Universal Robots URScript: 2024golden.script

def unnamed():
  set_tcp(p[0.0,0.0,0.0,0.0,0.0,0.0])
  set_standard_analog_input_domain(0, 1)
  set_standard_analog_input_domain(1, 1)
  set_tool_analog_input_domain(0, 1)
  set_tool_analog_input_domain(1, 1)
  set_analog_outputdomain(0, 0)
  set_analog_outputdomain(1, 0)
  set_input_actions_to_default()
  set_target_payload(1.070000, [0.002000, 0.003000, 0.057000], [0.001723, 0.001723, 0.001723, 0.000000, 0.000000, 0.000000])
  set_tool_communication(True, 1000000, 2, 1, 1.5, 3.5)
  set_tool_output_mode(0)
  set_tool_digital_output_mode(0, 1)
  set_tool_digital_output_mode(1, 1)
  set_tool_voltage(0)
  set_gravity([0.0, 0.0, 9.82])
  step_count_2c8ba0bd_3175_4124_8579_105621cd2361 = 0.0
  thread Step_Counter_Thread_abff76f1_d808_4649_b515_a114c75a653f():
    while (True):
      step_count_2c8ba0bd_3175_4124_8579_105621cd2361 = step_count_2c8ba0bd_3175_4124_8579_105621cd2361 + 1.0
      sync()
    end
  end
  run Step_Counter_Thread_abff76f1_d808_4649_b515_a114c75a653f()
  set_safety_mode_transition_hardness(1)
  global Plane_1=p[-0.700006141123905,1.3454883874109249E-6,0.3910559577028425,-1.2089868272251132,-1.2089999932245832,1.20858562628424]
  global Plane_2=p[0.0,0.0,0.0,0.0,0.0,0.0]
  global Point_1=p[0.6913645118948067,-0.12399382748223003,0.49223711947071,-1.2983729986843258,1.1259514972191385,-1.2203503861141718]
  $ 1 "Robot Program"
  $ 2 "Script: 2024Dragon_V2_golden_pen.script"
  def Machining1():
    # Default parameters:
    global speed_ms = 0.3
    global speed_rads = 0.75
    global accel_mss = 3
    global accel_radss = 1.2
    global blend_radius_m = 0.001

    # Add subprograms here
    # Start of main program
    # Program generated by RoboDK v5.6.5 for UR10e on 10/01/2024 17:37:16
    # Using nominal kinematics.
    blend_radius_m = 0.001
    speed_ms = 1.000
    # set_reference(p[0.320000, -0.152000, -0.013500, 0.000000, 0.000000, 0.000000])
    set_tcp(p[0.000000, 0.000000, 0.252000, 0.000000, 0.000000, 0.000000])
    # Show Tool
    movej([0.070455, -1.056852, -2.625487, -1.030050, 1.570796, 1.641252],accel_radss,speed_rads,0,blend_radius_m)
    movel([0.070455, -1.056852, -2.625487, -1.030050, 1.570796, 1.641252],accel_mss,speed_ms,0,blend_radius_m)
    # Splitting Linear movement in 32 (instruction 7: MoveL 3)
    movel([0.070455, -1.058454, -2.626785, -1.027150, 1.570796, 1.641252],accel_mss,speed_ms,0,blend_radius_m)
    movel([0.070455, -1.060067, -2.628081, -1.024241, 1.570796, 1.641252],accel_mss,speed_ms,0,blend_radius_m)
    movel([0.070455, -1.061692, -2.629375, -1.021322, 1.570796, 1.641252],accel_mss,speed_ms,0,blend_radius_m)
    movel([0.070455, -1.063329, -2.630667, -1.018394, 1.570796, 1.641252],accel_mss,speed_ms,0,blend_radius_m)
    movel([0.070455, -1.064977, -2.631956, -1.015456, 1.570796, 1.641252],accel_mss,speed_ms,0,blend_radius_m)
    movel([0.070455, -1.066637, -2.633243, -1.012509, 1.570796, 1.641252],accel_mss,speed_ms,0,blend_radius_m)
    movel([0.070455, -1.068308, -2.634528, -1.009553, 1.570796, 1.641252],accel_mss,speed_ms,0,blend_radius_m)
    movel([0.070455, -1.069991, -2.635811, -1.006586, 1.570796, 1.641252],accel_mss,speed_ms,0,blend_radius_m)
    movel([0.070455, -1.071686, -2.637092, -1.003611, 1.570796, 1.641252],accel_mss,speed_ms,0,blend_radius_m)
    movel([0.070455, -1.073393, -2.638371, -1.000625, 1.570796, 1.641252],accel_mss,speed_ms,0,blend_radius_m)
    movel([0.070455, -1.075112, -2.639647, -0.997630, 1.570796, 1.641252],accel_mss,speed_ms,0,blend_radius_m)
    movel([0.070455, -1.076843, -2.640921, -0.994625, 1.570796, 1.641252],accel_mss,speed_ms,0,blend_radius_m)
    movel([0.070455, -1.078586, -2.642192, -0.991611, 1.570796, 1.641252],accel_mss,speed_ms,0,blend_radius_m)
    movel([0.070455, -1.080341, -2.643462, -0.988586, 1.570796, 1.641252],accel_mss,speed_ms,0,blend_radius_m)
    movel([0.070455, -1.082109, -2.644729, -0.985551, 1.570796, 1.641252],accel_mss,speed_ms,0,blend_radius_m)
    movel([0.070455, -1.083888, -2.645994, -0.982507, 1.570796, 1.641252],accel_mss,speed_ms,0,blend_radius_m)
    movel([0.070455, -1.085680, -2.647256, -0.979453, 1.570796, 1.641252],accel_mss,speed_ms,0,blend_radius_m)
    movel([0.070455, -1.087485, -2.648516, -0.976388, 1.570796, 1.641252],accel_mss,speed_ms,0,blend_radius_m)
    movel([0.070455, -1.089301, -2.649774, -0.973313, 1.570796, 1.641252],accel_mss,speed_ms,0,blend_radius_m)
    movel([0.070455, -1.091131, -2.651030, -0.970229, 1.570796, 1.641252],accel_mss,speed_ms,0,blend_radius_m)
    movel([0.070455, -1.092973, -2.652283, -0.967134, 1.570796, 1.641252],accel_mss,speed_ms,0,blend_radius_m)
    movel([0.070455, -1.094827, -2.653533, -0.964028, 1.570796, 1.641252],accel_mss,speed_ms,0,blend_radius_m)
    movel([0.070455, -1.096695, -2.654781, -0.960913, 1.570796, 1.641252],accel_mss,speed_ms,0,blend_radius_m)
    movel([0.070455, -1.098575, -2.656027, -0.957787, 1.570796, 1.641252],accel_mss,speed_ms,0,blend_radius_m)
    movel([0.070455, -1.100468, -2.657271, -0.954651, 1.570796, 1.641252],accel_mss,speed_ms,0,blend_radius_m)
    movel([0.070455, -1.102374, -2.658511, -0.951504, 1.570796, 1.641252],accel_mss,speed_ms,0,blend_radius_m)
    movel([0.070455, -1.104293, -2.659750, -0.948346, 1.570796, 1.641252],accel_mss,speed_ms,0,blend_radius_m)
    movel([0.070455, -1.106224, -2.660986, -0.945179, 1.570796, 1.641252],accel_mss,speed_ms,0,blend_radius_m)
    movel([0.070455, -1.108170, -2.662219, -0.942000, 1.570796, 1.641252],accel_mss,speed_ms,0,blend_radius_m)
    movel([0.070455, -1.110128, -2.663450, -0.938811, 1.570796, 1.641252],accel_mss,speed_ms,0,blend_radius_m)
    movel([0.070455, -1.112099, -2.664678, -0.935611, 1.570796, 1.641252],accel_mss,speed_ms,0,blend_radius_m)
    movel([0.070455, -1.114084, -2.665904, -0.932401, 1.570796, 1.641252],accel_mss,speed_ms,0,blend_radius_m)
    movel([0.070455, -1.114084, -2.665904, -0.932401, 1.570796, 1.641252],accel_mss,speed_ms,0,blend_radius_m)
    speed_ms = 1.000
    movel([0.070455, -1.114084, -2.665904, -0.932401, 1.570796, 1.641252],accel_mss,speed_ms,0,blend_radius_m)
    movel([0.070455, -1.114084, -2.665904, -0.932401, 1.570796, 1.641252],accel_mss,speed_ms,0,blend_radius_m)
    movel([0.070455, -1.114084, -2.665904, -0.932401, 1.570796, 1.641252],accel_mss,speed_ms,0,blend_radius_m)
    speed_ms = 0.005
    # Splitting Linear movement in 22 (instruction 14: MoveL 8)
    movel([0.070455, -1.112159, -2.664716, -0.935514, 1.570796, 1.641252],accel_mss,speed_ms,0,blend_radius_m)
    movel([0.070455, -1.110247, -2.663525, -0.938618, 1.570796, 1.641252],accel_mss,speed_ms,0,blend_radius_m)
    movel([0.070455, -1.108347, -2.662331, -0.941711, 1.570796, 1.641252],accel_mss,speed_ms,0,blend_radius_m)
    movel([0.070455, -1.106460, -2.661135, -0.944794, 1.570796, 1.641252],accel_mss,speed_ms,0,blend_radius_m)
    movel([0.070455, -1.104584, -2.659937, -0.947867, 1.570796, 1.641252],accel_mss,speed_ms,0,blend_radius_m)
    movel([0.070455, -1.102722, -2.658737, -0.950930, 1.570796, 1.641252],accel_mss,speed_ms,0,blend_radius_m)
    movel([0.070455, -1.100871, -2.657534, -0.953984, 1.570796, 1.641252],accel_mss,speed_ms,0,blend_radius_m)
    movel([0.070455, -1.099033, -2.656329, -0.957027, 1.570796, 1.641252],accel_mss,speed_ms,0,blend_radius_m)
    movel([0.070455, -1.097206, -2.655121, -0.960061, 1.570796, 1.641252],accel_mss,speed_ms,0,blend_radius_m)
    movel([0.070455, -1.095392, -2.653912, -0.963085, 1.570796, 1.641252],accel_mss,speed_ms,0,blend_radius_m)
    movel([0.070455, -1.093590, -2.652700, -0.966100, 1.570796, 1.641252],accel_mss,speed_ms,0,blend_radius_m)
    movel([0.070455, -1.091799, -2.651486, -0.969104, 1.570796, 1.641252],accel_mss,speed_ms,0,blend_radius_m)
    movel([0.070455, -1.090021, -2.650269, -0.972099, 1.570796, 1.641252],accel_mss,speed_ms,0,blend_radius_m)
    movel([0.070455, -1.088254, -2.649050, -0.975085, 1.570796, 1.641252],accel_mss,speed_ms,0,blend_radius_m)
    movel([0.070455, -1.086499, -2.647829, -0.978061, 1.570796, 1.641252],accel_mss,speed_ms,0,blend_radius_m)
    movel([0.070455, -1.084755, -2.646606, -0.981027, 1.570796, 1.641252],accel_mss,speed_ms,0,blend_radius_m)
    movel([0.070455, -1.083024, -2.645381, -0.983984, 1.570796, 1.641252],accel_mss,speed_ms,0,blend_radius_m)
    movel([0.070455, -1.081304, -2.644153, -0.986932, 1.570796, 1.641252],accel_mss,speed_ms,0,blend_radius_m)
    movel([0.070455, -1.079595, -2.642924, -0.989870, 1.570796, 1.641252],accel_mss,speed_ms,0,blend_radius_m)
    movel([0.070455, -1.077898, -2.641692, -0.992799, 1.570796, 1.641252],accel_mss,speed_ms,0,blend_radius_m)
    movel([0.070455, -1.076212, -2.640458, -0.995719, 1.570796, 1.641252],accel_mss,speed_ms,0,blend_radius_m)
    movel([0.070455, -1.074538, -2.639222, -0.998630, 1.570796, 1.641252],accel_mss,speed_ms,0,blend_radius_m)
    speed_ms = 1.000
    # Splitting Linear movement in 22 (instruction 16: MoveL 9)
    movel([0.070455, -1.076212, -2.640458, -0.995719, 1.570796, 1.641252],accel_mss,speed_ms,0,blend_radius_m)
    movel([0.070455, -1.077898, -2.641692, -0.992799, 1.570796, 1.641252],accel_mss,speed_ms,0,blend_radius_m)
    movel([0.070455, -1.079595, -2.642924, -0.989870, 1.570796, 1.641252],accel_mss,speed_ms,0,blend_radius_m)
    movel([0.070455, -1.081304, -2.644153, -0.986932, 1.570796, 1.641252],accel_mss,speed_ms,0,blend_radius_m)
    movel([0.070455, -1.083024, -2.645381, -0.983984, 1.570796, 1.641252],accel_mss,speed_ms,0,blend_radius_m)
    movel([0.070455, -1.084755, -2.646606, -0.981027, 1.570796, 1.641252],accel_mss,speed_ms,0,blend_radius_m)
    movel([0.070455, -1.086499, -2.647829, -0.978061, 1.570796, 1.641252],accel_mss,speed_ms,0,blend_radius_m)
    movel([0.070455, -1.088254, -2.649050, -0.975085, 1.570796, 1.641252],accel_mss,speed_ms,0,blend_radius_m)
    movel([0.070455, -1.090021, -2.650269, -0.972099, 1.570796, 1.641252],accel_mss,speed_ms,0,blend_radius_m)
    movel([0.070455, -1.091799, -2.651486, -0.969104, 1.570796, 1.641252],accel_mss,speed_ms,0,blend_radius_m)
    movel([0.070455, -1.093590, -2.652700, -0.966100, 1.570796, 1.641252],accel_mss,speed_ms,0,blend_radius_m)
    movel([0.070455, -1.095392, -2.653912, -0.963085, 1.570796, 1.641252],accel_mss,speed_ms,0,blend_radius_m)
    movel([0.070455, -1.097206, -2.655121, -0.960061, 1.570796, 1.641252],accel_mss,speed_ms,0,blend_radius_m)
    movel([0.070455, -1.099033, -2.656329, -0.957027, 1.570796, 1.641252],accel_mss,speed_ms,0,blend_radius_m)
    movel([0.070455, -1.100871, -2.657534, -0.953984, 1.570796, 1.641252],accel_mss,speed_ms,0,blend_radius_m)
    movel([0.070455, -1.102722, -2.658737, -0.950930, 1.570796, 1.641252],accel_mss,speed_ms,0,blend_radius_m)
    movel([0.070455, -1.104584, -2.659937, -0.947867, 1.570796, 1.641252],accel_mss,speed_ms,0,blend_radius_m)
    movel([0.070455, -1.106460, -2.661135, -0.944794, 1.570796, 1.641252],accel_mss,speed_ms,0,blend_radius_m)
    movel([0.070455, -1.108347, -2.662331, -0.941711, 1.570796, 1.641252],accel_mss,speed_ms,0,blend_radius_m)
    movel([0.070455, -1.110247, -2.663525, -0.938618, 1.570796, 1.641252],accel_mss,speed_ms,0,blend_radius_m)
    movel([0.070455, -1.112159, -2.664716, -0.935514, 1.570796, 1.641252],accel_mss,speed_ms,0,blend_radius_m)
    movel([0.070455, -1.114084, -2.665904, -0.932401, 1.570796, 1.641252],accel_mss,speed_ms,0,blend_radius_m)
    speed_ms = 0.040
    movel([0.070455, -1.114084, -2.665904, -0.932401, 1.570796, 1.641252],accel_mss,speed_ms,0,blend_radius_m)
    speed_ms = 1.000
    movel([0.070455, -1.114084, -2.665904, -0.932401, 1.570796, 1.641252],accel_mss,speed_ms,0,blend_radius_m)
    # Splitting Linear movement in 152 (instruction 21: MoveL 12)
    movel([0.070832, -1.116719, -2.664817, -0.930853, 1.570796, 1.641628],accel_mss,speed_ms,0,blend_radius_m)
    movel([0.071206, -1.119347, -2.663727, -0.929315, 1.570796, 1.642002],accel_mss,speed_ms,0,blend_radius_m)
    movel([0.071578, -1.121968, -2.662633, -0.927788, 1.570796, 1.642374],accel_mss,speed_ms,0,blend_radius_m)
    movel([0.071947, -1.124581, -2.661536, -0.926272, 1.570796, 1.642743],accel_mss,speed_ms,0,blend_radius_m)
    movel([0.072314, -1.127187, -2.660435, -0.924767, 1.570796, 1.643111],accel_mss,speed_ms,0,blend_radius_m)
    movel([0.072679, -1.129786, -2.659331, -0.923272, 1.570796, 1.643476],accel_mss,speed_ms,0,blend_radius_m)
    movel([0.073042, -1.132378, -2.658223, -0.921788, 1.570796, 1.643839],accel_mss,speed_ms,0,blend_radius_m)
    movel([0.073403, -1.134962, -2.657112, -0.920315, 1.570796, 1.644199],accel_mss,speed_ms,0,blend_radius_m)
    movel([0.073761, -1.137540, -2.655997, -0.918852, 1.570796, 1.644558],accel_mss,speed_ms,0,blend_radius_m)
    movel([0.074117, -1.140110, -2.654879, -0.917400, 1.570796, 1.644914],accel_mss,speed_ms,0,blend_radius_m)
    movel([0.074472, -1.142673, -2.653758, -0.915958, 1.570796, 1.645268],accel_mss,speed_ms,0,blend_radius_m)
    movel([0.074824, -1.145229, -2.652633, -0.914527, 1.570796, 1.645620],accel_mss,speed_ms,0,blend_radius_m)
    movel([0.075173, -1.147778, -2.651505, -0.913106, 1.570796, 1.645970],accel_mss,speed_ms,0,blend_radius_m)
    movel([0.075521, -1.150320, -2.650374, -0.911695, 1.570796, 1.646318],accel_mss,speed_ms,0,blend_radius_m)
    movel([0.075867, -1.152855, -2.649239, -0.910295, 1.570796, 1.646663],accel_mss,speed_ms,0,blend_radius_m)
    movel([0.076211, -1.155382, -2.648101, -0.908905, 1.570796, 1.647007],accel_mss,speed_ms,0,blend_radius_m)
    movel([0.076552, -1.157903, -2.646960, -0.907526, 1.570796, 1.647349],accel_mss,speed_ms,0,blend_radius_m)
    movel([0.076892, -1.160417, -2.645816, -0.906157, 1.570796, 1.647688],accel_mss,speed_ms,0,blend_radius_m)
    movel([0.077230, -1.162924, -2.644668, -0.904797, 1.570796, 1.648026],accel_mss,speed_ms,0,blend_radius_m)
    movel([0.077565, -1.165423, -2.643517, -0.903448, 1.570796, 1.648362],accel_mss,speed_ms,0,blend_radius_m)
    movel([0.077899, -1.167916, -2.642363, -0.902110, 1.570796, 1.648695],accel_mss,speed_ms,0,blend_radius_m)
    movel([0.078231, -1.170402, -2.641206, -0.900781, 1.570796, 1.649027],accel_mss,speed_ms,0,blend_radius_m)
    movel([0.078561, -1.172882, -2.640045, -0.899462, 1.570796, 1.649357],accel_mss,speed_ms,0,blend_radius_m)
    movel([0.078888, -1.175354, -2.638882, -0.898153, 1.570796, 1.649685],accel_mss,speed_ms,0,blend_radius_m)
    movel([0.079214, -1.177819, -2.637715, -0.896855, 1.570796, 1.650011],accel_mss,speed_ms,0,blend_radius_m)
    movel([0.079539, -1.180278, -2.636545, -0.895566, 1.570796, 1.650335],accel_mss,speed_ms,0,blend_radius_m)
    movel([0.079861, -1.182730, -2.635372, -0.894287, 1.570796, 1.650657],accel_mss,speed_ms,0,blend_radius_m)
    movel([0.080181, -1.185175, -2.634196, -0.893018, 1.570796, 1.650978],accel_mss,speed_ms,0,blend_radius_m)
    movel([0.080500, -1.187614, -2.633017, -0.891758, 1.570796, 1.651296],accel_mss,speed_ms,0,blend_radius_m)
    movel([0.080817, -1.190045, -2.631835, -0.890509, 1.570796, 1.651613],accel_mss,speed_ms,0,blend_radius_m)
    movel([0.081131, -1.192470, -2.630650, -0.889269, 1.570796, 1.651928],accel_mss,speed_ms,0,blend_radius_m)
    movel([0.081445, -1.194889, -2.629461, -0.888039, 1.570796, 1.652241],accel_mss,speed_ms,0,blend_radius_m)
    movel([0.081756, -1.197300, -2.628270, -0.886818, 1.570796, 1.652552],accel_mss,speed_ms,0,blend_radius_m)
    movel([0.082066, -1.199706, -2.627076, -0.885608, 1.570796, 1.652862],accel_mss,speed_ms,0,blend_radius_m)
    movel([0.082374, -1.202104, -2.625879, -0.884406, 1.570796, 1.653170],accel_mss,speed_ms,0,blend_radius_m)
    movel([0.082680, -1.204496, -2.624679, -0.883214, 1.570796, 1.653476],accel_mss,speed_ms,0,blend_radius_m)
    movel([0.082984, -1.206881, -2.623475, -0.882032, 1.570796, 1.653780],accel_mss,speed_ms,0,blend_radius_m)
    movel([0.083287, -1.209260, -2.622269, -0.880859, 1.570796, 1.654083],accel_mss,speed_ms,0,blend_radius_m)
    movel([0.083588, -1.211633, -2.621060, -0.879696, 1.570796, 1.654384],accel_mss,speed_ms,0,blend_radius_m)
    movel([0.083887, -1.213999, -2.619848, -0.878542, 1.570796, 1.654684],accel_mss,speed_ms,0,blend_radius_m)
    movel([0.084185, -1.216359, -2.618634, -0.877397, 1.570796, 1.654981],accel_mss,speed_ms,0,blend_radius_m)
    movel([0.084481, -1.218712, -2.617416, -0.876261, 1.570796, 1.655277],accel_mss,speed_ms,0,blend_radius_m)
    movel([0.084775, -1.221058, -2.616196, -0.875135, 1.570796, 1.655572],accel_mss,speed_ms,0,blend_radius_m)
    movel([0.085068, -1.223399, -2.614972, -0.874018, 1.570796, 1.655864],accel_mss,speed_ms,0,blend_radius_m)
    movel([0.085359, -1.225733, -2.613746, -0.872910, 1.570796, 1.656156],accel_mss,speed_ms,0,blend_radius_m)
    movel([0.085649, -1.228061, -2.612517, -0.871811, 1.570796, 1.656445],accel_mss,speed_ms,0,blend_radius_m)
    movel([0.085937, -1.230382, -2.611285, -0.870721, 1.570796, 1.656733],accel_mss,speed_ms,0,blend_radius_m)
    movel([0.086223, -1.232698, -2.610051, -0.869641, 1.570796, 1.657020],accel_mss,speed_ms,0,blend_radius_m)
    movel([0.086508, -1.235007, -2.608813, -0.868569, 1.570796, 1.657304],accel_mss,speed_ms,0,blend_radius_m)
    movel([0.086791, -1.237310, -2.607573, -0.867506, 1.570796, 1.657588],accel_mss,speed_ms,0,blend_radius_m)
    movel([0.087073, -1.239606, -2.606330, -0.866452, 1.570796, 1.657869],accel_mss,speed_ms,0,blend_radius_m)
    movel([0.087353, -1.241897, -2.605085, -0.865407, 1.570796, 1.658150],accel_mss,speed_ms,0,blend_radius_m)
    movel([0.087632, -1.244181, -2.603836, -0.864371, 1.570796, 1.658428],accel_mss,speed_ms,0,blend_radius_m)
    movel([0.087909, -1.246460, -2.602585, -0.863344, 1.570796, 1.658706],accel_mss,speed_ms,0,blend_radius_m)
    movel([0.088185, -1.248732, -2.601332, -0.862325, 1.570796, 1.658981],accel_mss,speed_ms,0,blend_radius_m)
    movel([0.088459, -1.250998, -2.600075, -0.861315, 1.570796, 1.659256],accel_mss,speed_ms,0,blend_radius_m)
    movel([0.088732, -1.253259, -2.598816, -0.860314, 1.570796, 1.659528],accel_mss,speed_ms,0,blend_radius_m)
    movel([0.089004, -1.255513, -2.597555, -0.859322, 1.570796, 1.659800],accel_mss,speed_ms,0,blend_radius_m)
    movel([0.089273, -1.257761, -2.596290, -0.858338, 1.570796, 1.660070],accel_mss,speed_ms,0,blend_radius_m)
    movel([0.089542, -1.260004, -2.595023, -0.857362, 1.570796, 1.660338],accel_mss,speed_ms,0,blend_radius_m)
    movel([0.089809, -1.262240, -2.593754, -0.856395, 1.570796, 1.660605],accel_mss,speed_ms,0,blend_radius_m)
    movel([0.090075, -1.264471, -2.592482, -0.855437, 1.570796, 1.660871],accel_mss,speed_ms,0,blend_radius_m)
    movel([0.090339, -1.266695, -2.591207, -0.854487, 1.570796, 1.661135],accel_mss,speed_ms,0,blend_radius_m)
    movel([0.090602, -1.268914, -2.589929, -0.853545, 1.570796, 1.661398],accel_mss,speed_ms,0,blend_radius_m)
    movel([0.090863, -1.271127, -2.588650, -0.852612, 1.570796, 1.661660],accel_mss,speed_ms,0,blend_radius_m)
    movel([0.091123, -1.273335, -2.587367, -0.851687, 1.570796, 1.661920],accel_mss,speed_ms,0,blend_radius_m)
    movel([0.091382, -1.275537, -2.586082, -0.850770, 1.570796, 1.662178],accel_mss,speed_ms,0,blend_radius_m)
    movel([0.091640, -1.277732, -2.584795, -0.849862, 1.570796, 1.662436],accel_mss,speed_ms,0,blend_radius_m)
    movel([0.091896, -1.279923, -2.583505, -0.848962, 1.570796, 1.662692],accel_mss,speed_ms,0,blend_radius_m)
    movel([0.092150, -1.282107, -2.582212, -0.848070, 1.570796, 1.662947],accel_mss,speed_ms,0,blend_radius_m)
    movel([0.092404, -1.284286, -2.580917, -0.847186, 1.570796, 1.663200],accel_mss,speed_ms,0,blend_radius_m)
    movel([0.092656, -1.286460, -2.579620, -0.846310, 1.570796, 1.663452],accel_mss,speed_ms,0,blend_radius_m)
    movel([0.092907, -1.288627, -2.578320, -0.845442, 1.570796, 1.663703],accel_mss,speed_ms,0,blend_radius_m)
    movel([0.093156, -1.290790, -2.577017, -0.844582, 1.570796, 1.663953],accel_mss,speed_ms,0,blend_radius_m)
    movel([0.093405, -1.292946, -2.575712, -0.843730, 1.570796, 1.664201],accel_mss,speed_ms,0,blend_radius_m)
    movel([0.093652, -1.295097, -2.574405, -0.842886, 1.570796, 1.664448],accel_mss,speed_ms,0,blend_radius_m)
    movel([0.093897, -1.297243, -2.573095, -0.842050, 1.570796, 1.664694],accel_mss,speed_ms,0,blend_radius_m)
    movel([0.094142, -1.299383, -2.571783, -0.841222, 1.570796, 1.664938],accel_mss,speed_ms,0,blend_radius_m)
    movel([0.094385, -1.301518, -2.570469, -0.840402, 1.570796, 1.665182],accel_mss,speed_ms,0,blend_radius_m)
    movel([0.094627, -1.303648, -2.569152, -0.839589, 1.570796, 1.665424],accel_mss,speed_ms,0,blend_radius_m)
    movel([0.094868, -1.305772, -2.567833, -0.838784, 1.570796, 1.665664],accel_mss,speed_ms,0,blend_radius_m)
    movel([0.095108, -1.307891, -2.566511, -0.837987, 1.570796, 1.665904],accel_mss,speed_ms,0,blend_radius_m)
    movel([0.095346, -1.310004, -2.565187, -0.837198, 1.570796, 1.666142],accel_mss,speed_ms,0,blend_radius_m)
    movel([0.095583, -1.312112, -2.563861, -0.836416, 1.570796, 1.666380],accel_mss,speed_ms,0,blend_radius_m)
    movel([0.095819, -1.314215, -2.562532, -0.835642, 1.570796, 1.666616],accel_mss,speed_ms,0,blend_radius_m)
    movel([0.096054, -1.316313, -2.561201, -0.834875, 1.570796, 1.666851],accel_mss,speed_ms,0,blend_radius_m)
    movel([0.096288, -1.318405, -2.559868, -0.834116, 1.570796, 1.667084],accel_mss,speed_ms,0,blend_radius_m)
    movel([0.096520, -1.320492, -2.558533, -0.833364, 1.570796, 1.667317],accel_mss,speed_ms,0,blend_radius_m)
    movel([0.096752, -1.322575, -2.557195, -0.832620, 1.570796, 1.667548],accel_mss,speed_ms,0,blend_radius_m)
    movel([0.096982, -1.324652, -2.555855, -0.831883, 1.570796, 1.667778],accel_mss,speed_ms,0,blend_radius_m)
    movel([0.097211, -1.326723, -2.554512, -0.831153, 1.570796, 1.668007],accel_mss,speed_ms,0,blend_radius_m)
    movel([0.097439, -1.328790, -2.553168, -0.830431, 1.570796, 1.668235],accel_mss,speed_ms,0,blend_radius_m)
    movel([0.097666, -1.330852, -2.551821, -0.829716, 1.570796, 1.668462],accel_mss,speed_ms,0,blend_radius_m)
    movel([0.097892, -1.332909, -2.550472, -0.829009, 1.570796, 1.668688],accel_mss,speed_ms,0,blend_radius_m)
    movel([0.098116, -1.334960, -2.549120, -0.828308, 1.570796, 1.668913],accel_mss,speed_ms,0,blend_radius_m)
    movel([0.098340, -1.337007, -2.547767, -0.827615, 1.570796, 1.669136],accel_mss,speed_ms,0,blend_radius_m)
    movel([0.098562, -1.339049, -2.546411, -0.826929, 1.570796, 1.669359],accel_mss,speed_ms,0,blend_radius_m)
    movel([0.098784, -1.341086, -2.545053, -0.826250, 1.570796, 1.669580],accel_mss,speed_ms,0,blend_radius_m)
    movel([0.099004, -1.343118, -2.543693, -0.825578, 1.570796, 1.669800],accel_mss,speed_ms,0,blend_radius_m)
    movel([0.099223, -1.345145, -2.542331, -0.824913, 1.570796, 1.670020],accel_mss,speed_ms,0,blend_radius_m)
    movel([0.099441, -1.347167, -2.540966, -0.824256, 1.570796, 1.670238],accel_mss,speed_ms,0,blend_radius_m)
    movel([0.099659, -1.349185, -2.539600, -0.823605, 1.570796, 1.670455],accel_mss,speed_ms,0,blend_radius_m)
    movel([0.099875, -1.351197, -2.538231, -0.822961, 1.570796, 1.670671],accel_mss,speed_ms,0,blend_radius_m)
    movel([0.100090, -1.353205, -2.536860, -0.822324, 1.570796, 1.670886],accel_mss,speed_ms,0,blend_radius_m)
    movel([0.100304, -1.355208, -2.535487, -0.821694, 1.570796, 1.671100],accel_mss,speed_ms,0,blend_radius_m)
    movel([0.100517, -1.357207, -2.534112, -0.821070, 1.570796, 1.671313],accel_mss,speed_ms,0,blend_radius_m)
    movel([0.100729, -1.359200, -2.532735, -0.820454, 1.570796, 1.671525],accel_mss,speed_ms,0,blend_radius_m)
    movel([0.100940, -1.361189, -2.531355, -0.819844, 1.570796, 1.671736],accel_mss,speed_ms,0,blend_radius_m)
    movel([0.101150, -1.363174, -2.529974, -0.819241, 1.570796, 1.671946],accel_mss,speed_ms,0,blend_radius_m)
    movel([0.101359, -1.365154, -2.528590, -0.818645, 1.570796, 1.672155],accel_mss,speed_ms,0,blend_radius_m)
    movel([0.101567, -1.367129, -2.527205, -0.818055, 1.570796, 1.672363],accel_mss,speed_ms,0,blend_radius_m)
    movel([0.101774, -1.369099, -2.525817, -0.817473, 1.570796, 1.672570],accel_mss,speed_ms,0,blend_radius_m)
    movel([0.101980, -1.371065, -2.524427, -0.816896, 1.570796, 1.672776],accel_mss,speed_ms,0,blend_radius_m)
    movel([0.102185, -1.373027, -2.523036, -0.816326, 1.570796, 1.672981],accel_mss,speed_ms,0,blend_radius_m)
    movel([0.102389, -1.374984, -2.521642, -0.815763, 1.570796, 1.673186],accel_mss,speed_ms,0,blend_radius_m)
    movel([0.102593, -1.376937, -2.520246, -0.815206, 1.570796, 1.673389],accel_mss,speed_ms,0,blend_radius_m)
    movel([0.102795, -1.378885, -2.518848, -0.814656, 1.570796, 1.673591],accel_mss,speed_ms,0,blend_radius_m)
    movel([0.102996, -1.380828, -2.517448, -0.814112, 1.570796, 1.673792],accel_mss,speed_ms,0,blend_radius_m)
    movel([0.103197, -1.382768, -2.516046, -0.813575, 1.570796, 1.673993],accel_mss,speed_ms,0,blend_radius_m)
    movel([0.103396, -1.384703, -2.514642, -0.813044, 1.570796, 1.674192],accel_mss,speed_ms,0,blend_radius_m)
    movel([0.103595, -1.386633, -2.513237, -0.812519, 1.570796, 1.674391],accel_mss,speed_ms,0,blend_radius_m)
    movel([0.103792, -1.388559, -2.511829, -0.812001, 1.570796, 1.674588],accel_mss,speed_ms,0,blend_radius_m)
    movel([0.103989, -1.390481, -2.510419, -0.811489, 1.570796, 1.674785],accel_mss,speed_ms,0,blend_radius_m)
    movel([0.104185, -1.392399, -2.509007, -0.810983, 1.570796, 1.674981],accel_mss,speed_ms,0,blend_radius_m)
    movel([0.104380, -1.394312, -2.507593, -0.810483, 1.570796, 1.675176],accel_mss,speed_ms,0,blend_radius_m)
    movel([0.104574, -1.396221, -2.506178, -0.809990, 1.570796, 1.675370],accel_mss,speed_ms,0,blend_radius_m)
    movel([0.104767, -1.398126, -2.504760, -0.809503, 1.570796, 1.675563],accel_mss,speed_ms,0,blend_radius_m)
    movel([0.104959, -1.400027, -2.503341, -0.809022, 1.570796, 1.675755],accel_mss,speed_ms,0,blend_radius_m)
    movel([0.105151, -1.401923, -2.501919, -0.808546, 1.570796, 1.675947],accel_mss,speed_ms,0,blend_radius_m)
    movel([0.105341, -1.403816, -2.500496, -0.808077, 1.570796, 1.676137],accel_mss,speed_ms,0,blend_radius_m)
    movel([0.105531, -1.405704, -2.499070, -0.807615, 1.570796, 1.676327],accel_mss,speed_ms,0,blend_radius_m)
    movel([0.105720, -1.407588, -2.497643, -0.807158, 1.570796, 1.676516],accel_mss,speed_ms,0,blend_radius_m)
    movel([0.105908, -1.409468, -2.496214, -0.806707, 1.570796, 1.676704],accel_mss,speed_ms,0,blend_radius_m)
    movel([0.106095, -1.411344, -2.494783, -0.806262, 1.570796, 1.676891],accel_mss,speed_ms,0,blend_radius_m)
    movel([0.106281, -1.413216, -2.493350, -0.805822, 1.570796, 1.677077],accel_mss,speed_ms,0,blend_radius_m)
    movel([0.106466, -1.415084, -2.491915, -0.805389, 1.570796, 1.677263],accel_mss,speed_ms,0,blend_radius_m)
    movel([0.106651, -1.416948, -2.490479, -0.804962, 1.570796, 1.677447],accel_mss,speed_ms,0,blend_radius_m)
    movel([0.106835, -1.418808, -2.489040, -0.804540, 1.570796, 1.677631],accel_mss,speed_ms,0,blend_radius_m)
    movel([0.107018, -1.420664, -2.487600, -0.804125, 1.570796, 1.677814],accel_mss,speed_ms,0,blend_radius_m)
    movel([0.107200, -1.422517, -2.486158, -0.803715, 1.570796, 1.677997],accel_mss,speed_ms,0,blend_radius_m)
    movel([0.107382, -1.424365, -2.484714, -0.803310, 1.570796, 1.678178],accel_mss,speed_ms,0,blend_radius_m)
    movel([0.107562, -1.426209, -2.483268, -0.802912, 1.570796, 1.678359],accel_mss,speed_ms,0,blend_radius_m)
    movel([0.107742, -1.428050, -2.481820, -0.802519, 1.570796, 1.678538],accel_mss,speed_ms,0,blend_radius_m)
    movel([0.107921, -1.429887, -2.480371, -0.802132, 1.570796, 1.678717],accel_mss,speed_ms,0,blend_radius_m)
    movel([0.108099, -1.431719, -2.478919, -0.801750, 1.570796, 1.678896],accel_mss,speed_ms,0,blend_radius_m)
    movel([0.108277, -1.433548, -2.477466, -0.801374, 1.570796, 1.679073],accel_mss,speed_ms,0,blend_radius_m)
    movel([0.108453, -1.435374, -2.476011, -0.801004, 1.570796, 1.679250],accel_mss,speed_ms,0,blend_radius_m)
    movel([0.108629, -1.437195, -2.474555, -0.800639, 1.570796, 1.679426],accel_mss,speed_ms,0,blend_radius_m)
    movel([0.108804, -1.439013, -2.473096, -0.800280, 1.570796, 1.679601],accel_mss,speed_ms,0,blend_radius_m)
    movel([0.108979, -1.440827, -2.471636, -0.799926, 1.570796, 1.679775],accel_mss,speed_ms,0,blend_radius_m)
    movel([0.109152, -1.442638, -2.470174, -0.799578, 1.570796, 1.679949],accel_mss,speed_ms,0,blend_radius_m)
    movel([0.109325, -1.444445, -2.468710, -0.799235, 1.570796, 1.680122],accel_mss,speed_ms,0,blend_radius_m)
    speed_ms = 0.005
    # Splitting Linear movement in 22 (instruction 23: MoveL 13)
    movel([0.109325, -1.446108, -2.469581, -0.796700, 1.570796, 1.680122],accel_mss,speed_ms,0,blend_radius_m)
    movel([0.109325, -1.447777, -2.470449, -0.794163, 1.570796, 1.680122],accel_mss,speed_ms,0,blend_radius_m)
    movel([0.109325, -1.449453, -2.471314, -0.791622, 1.570796, 1.680122],accel_mss,speed_ms,0,blend_radius_m)
    movel([0.109325, -1.451135, -2.472177, -0.789077, 1.570796, 1.680122],accel_mss,speed_ms,0,blend_radius_m)
    movel([0.109325, -1.452822, -2.473037, -0.786530, 1.570796, 1.680122],accel_mss,speed_ms,0,blend_radius_m)
    movel([0.109325, -1.454517, -2.473893, -0.783979, 1.570796, 1.680122],accel_mss,speed_ms,0,blend_radius_m)
    movel([0.109325, -1.456217, -2.474747, -0.781425, 1.570796, 1.680122],accel_mss,speed_ms,0,blend_radius_m)
    movel([0.109325, -1.457923, -2.475598, -0.778868, 1.570796, 1.680122],accel_mss,speed_ms,0,blend_radius_m)
    movel([0.109325, -1.459636, -2.476446, -0.776307, 1.570796, 1.680122],accel_mss,speed_ms,0,blend_radius_m)
    movel([0.109325, -1.461354, -2.477291, -0.773743, 1.570796, 1.680122],accel_mss,speed_ms,0,blend_radius_m)
    movel([0.109325, -1.463079, -2.478134, -0.771176, 1.570796, 1.680122],accel_mss,speed_ms,0,blend_radius_m)
    movel([0.109325, -1.464810, -2.478973, -0.768606, 1.570796, 1.680122],accel_mss,speed_ms,0,blend_radius_m)
    movel([0.109325, -1.466547, -2.479809, -0.766032, 1.570796, 1.680122],accel_mss,speed_ms,0,blend_radius_m)
    movel([0.109325, -1.468291, -2.480643, -0.763455, 1.570796, 1.680122],accel_mss,speed_ms,0,blend_radius_m)
    movel([0.109325, -1.470040, -2.481473, -0.760875, 1.570796, 1.680122],accel_mss,speed_ms,0,blend_radius_m)
    movel([0.109325, -1.471796, -2.482301, -0.758292, 1.570796, 1.680122],accel_mss,speed_ms,0,blend_radius_m)
    movel([0.109325, -1.473558, -2.483125, -0.755706, 1.570796, 1.680122],accel_mss,speed_ms,0,blend_radius_m)
    movel([0.109325, -1.475326, -2.483947, -0.753116, 1.570796, 1.680122],accel_mss,speed_ms,0,blend_radius_m)
    movel([0.109325, -1.477101, -2.484765, -0.750523, 1.570796, 1.680122],accel_mss,speed_ms,0,blend_radius_m)
    movel([0.109325, -1.478881, -2.485581, -0.747927, 1.570796, 1.680122],accel_mss,speed_ms,0,blend_radius_m)
    movel([0.109325, -1.480668, -2.486394, -0.745328, 1.570796, 1.680122],accel_mss,speed_ms,0,blend_radius_m)
    movel([0.109325, -1.482461, -2.487203, -0.742725, 1.570796, 1.680122],accel_mss,speed_ms,0,blend_radius_m)
    speed_ms = 0.035
    movel([0.106390, -1.483374, -2.486416, -0.742598, 1.570796, 1.677187],accel_mss,speed_ms,0,blend_radius_m)
    movel([0.104973, -1.483689, -2.486145, -0.742555, 1.570796, 1.675769],accel_mss,speed_ms,0,blend_radius_m)
    movel([0.103601, -1.483876, -2.485984, -0.742529, 1.570796, 1.674397],accel_mss,speed_ms,0,blend_radius_m)
    movel([0.102288, -1.483917, -2.485949, -0.742523, 1.570796, 1.673084],accel_mss,speed_ms,0,blend_radius_m)
    movel([0.101045, -1.483786, -2.486061, -0.742541, 1.570796, 1.671842],accel_mss,speed_ms,0,blend_radius_m)
    movel([0.099883, -1.483460, -2.486343, -0.742586, 1.570796, 1.670680],accel_mss,speed_ms,0,blend_radius_m)
    movel([0.098812, -1.482915, -2.486812, -0.742662, 1.570796, 1.669608],accel_mss,speed_ms,0,blend_radius_m)
    movel([0.097838, -1.482134, -2.487484, -0.742771, 1.570796, 1.668635],accel_mss,speed_ms,0,blend_radius_m)
    movel([0.097119, -1.481229, -2.488261, -0.742899, 1.570796, 1.667915],accel_mss,speed_ms,0,blend_radius_m)
    movel([0.096647, -1.480212, -2.489133, -0.743044, 1.570796, 1.667444],accel_mss,speed_ms,0,blend_radius_m)
    movel([0.096406, -1.479088, -2.490095, -0.743206, 1.570796, 1.667202],accel_mss,speed_ms,0,blend_radius_m)
    movel([0.096389, -1.477870, -2.491135, -0.743384, 1.570796, 1.667185],accel_mss,speed_ms,0,blend_radius_m)
    movel([0.096585, -1.476565, -2.492247, -0.743577, 1.570796, 1.667381],accel_mss,speed_ms,0,blend_radius_m)
    movel([0.096979, -1.475186, -2.493419, -0.743784, 1.570796, 1.667776],accel_mss,speed_ms,0,blend_radius_m)
    movel([0.097567, -1.473739, -2.494646, -0.744004, 1.570796, 1.668363],accel_mss,speed_ms,0,blend_radius_m)
    movel([0.098140, -1.472611, -2.495599, -0.744178, 1.570796, 1.668937],accel_mss,speed_ms,0,blend_radius_m)
    movel([0.098807, -1.471519, -2.496521, -0.744349, 1.570796, 1.669603],accel_mss,speed_ms,0,blend_radius_m)
    movel([0.099565, -1.470465, -2.497409, -0.744515, 1.570796, 1.670362],accel_mss,speed_ms,0,blend_radius_m)
    movel([0.100412, -1.469452, -2.498261, -0.744676, 1.570796, 1.671208],accel_mss,speed_ms,0,blend_radius_m)
    movel([0.101347, -1.468480, -2.499077, -0.744833, 1.570796, 1.672143],accel_mss,speed_ms,0,blend_radius_m)
    movel([0.102367, -1.467551, -2.499854, -0.744983, 1.570796, 1.673163],accel_mss,speed_ms,0,blend_radius_m)
    movel([0.103473, -1.466670, -2.500592, -0.745128, 1.570796, 1.674269],accel_mss,speed_ms,0,blend_radius_m)
    movel([0.107265, -1.463979, -2.502835, -0.745576, 1.570796, 1.678061],accel_mss,speed_ms,0,blend_radius_m)
    movel([0.109584, -1.462028, -2.504453, -0.745907, 1.570796, 1.680380],accel_mss,speed_ms,0,blend_radius_m)
    movel([0.111609, -1.459985, -2.506143, -0.746261, 1.570796, 1.682406],accel_mss,speed_ms,0,blend_radius_m)
    movel([0.113340, -1.457843, -2.507907, -0.746638, 1.570796, 1.684137],accel_mss,speed_ms,0,blend_radius_m)
    movel([0.114773, -1.455602, -2.509746, -0.747041, 1.570796, 1.685569],accel_mss,speed_ms,0,blend_radius_m)
    movel([0.115901, -1.453259, -2.511659, -0.747470, 1.570796, 1.686697],accel_mss,speed_ms,0,blend_radius_m)
    movel([0.116721, -1.450812, -2.513650, -0.747927, 1.570796, 1.687517],accel_mss,speed_ms,0,blend_radius_m)
    movel([0.117230, -1.448261, -2.515714, -0.748414, 1.570796, 1.688027],accel_mss,speed_ms,0,blend_radius_m)
    movel([0.117388, -1.447579, -2.516265, -0.748546, 1.570796, 1.688184],accel_mss,speed_ms,0,blend_radius_m)
    movel([0.117692, -1.447062, -2.516681, -0.748646, 1.570796, 1.688488],accel_mss,speed_ms,0,blend_radius_m)
    movel([0.118214, -1.446684, -2.516985, -0.748719, 1.570796, 1.689011],accel_mss,speed_ms,0,blend_radius_m)
    movel([0.119019, -1.446420, -2.517198, -0.748771, 1.570796, 1.689815],accel_mss,speed_ms,0,blend_radius_m)
    movel([0.119828, -1.446303, -2.517292, -0.748794, 1.570796, 1.690624],accel_mss,speed_ms,0,blend_radius_m)
    movel([0.120369, -1.446404, -2.517211, -0.748774, 1.570796, 1.691165],accel_mss,speed_ms,0,blend_radius_m)
    movel([0.120635, -1.446784, -2.516905, -0.748700, 1.570796, 1.691431],accel_mss,speed_ms,0,blend_radius_m)
    movel([0.120635, -1.447496, -2.516332, -0.748562, 1.570796, 1.691431],accel_mss,speed_ms,0,blend_radius_m)
    movel([0.120005, -1.450425, -2.513963, -0.748001, 1.570796, 1.690801],accel_mss,speed_ms,0,blend_radius_m)
    movel([0.119559, -1.451846, -2.512810, -0.747733, 1.570796, 1.690356],accel_mss,speed_ms,0,blend_radius_m)
    movel([0.118418, -1.454596, -2.510569, -0.747224, 1.570796, 1.689214],accel_mss,speed_ms,0,blend_radius_m)
    movel([0.117722, -1.455927, -2.509480, -0.746982, 1.570796, 1.688518],accel_mss,speed_ms,0,blend_radius_m)
    movel([0.116082, -1.458505, -2.507363, -0.746521, 1.570796, 1.686878],accel_mss,speed_ms,0,blend_radius_m)
    movel([0.115138, -1.459754, -2.506334, -0.746301, 1.570796, 1.685935],accel_mss,speed_ms,0,blend_radius_m)
    movel([0.113008, -1.462173, -2.504334, -0.745882, 1.570796, 1.683804],accel_mss,speed_ms,0,blend_radius_m)
    movel([0.111821, -1.463346, -2.503361, -0.745682, 1.570796, 1.682617],accel_mss,speed_ms,0,blend_radius_m)
    movel([0.109208, -1.465618, -2.501469, -0.745301, 1.570796, 1.680005],accel_mss,speed_ms,0,blend_radius_m)
    movel([0.106281, -1.467799, -2.499647, -0.744943, 1.570796, 1.677078],accel_mss,speed_ms,0,blend_radius_m)
    movel([0.104993, -1.468779, -2.498826, -0.744784, 1.570796, 1.675790],accel_mss,speed_ms,0,blend_radius_m)
    movel([0.103770, -1.469868, -2.497911, -0.744610, 1.570796, 1.674567],accel_mss,speed_ms,0,blend_radius_m)
    movel([0.102637, -1.471028, -2.496935, -0.744426, 1.570796, 1.673433],accel_mss,speed_ms,0,blend_radius_m)
    movel([0.101614, -1.472219, -2.495930, -0.744239, 1.570796, 1.672410],accel_mss,speed_ms,0,blend_radius_m)
    movel([0.100892, -1.473213, -2.495090, -0.744085, 1.570796, 1.671688],accel_mss,speed_ms,0,blend_radius_m)
    movel([0.100333, -1.474192, -2.494262, -0.743935, 1.570796, 1.671129],accel_mss,speed_ms,0,blend_radius_m)
    movel([0.099937, -1.475151, -2.493449, -0.743789, 1.570796, 1.670734],accel_mss,speed_ms,0,blend_radius_m)
    movel([0.099701, -1.476082, -2.492658, -0.743649, 1.570796, 1.670497],accel_mss,speed_ms,0,blend_radius_m)
    movel([0.099625, -1.476985, -2.491889, -0.743515, 1.570796, 1.670421],accel_mss,speed_ms,0,blend_radius_m)
    movel([0.099708, -1.477854, -2.491149, -0.743386, 1.570796, 1.670504],accel_mss,speed_ms,0,blend_radius_m)
    movel([0.099948, -1.478682, -2.490442, -0.743265, 1.570796, 1.670745],accel_mss,speed_ms,0,blend_radius_m)
    movel([0.100345, -1.479468, -2.489770, -0.743151, 1.570796, 1.671142],accel_mss,speed_ms,0,blend_radius_m)
    movel([0.100864, -1.480107, -2.489223, -0.743059, 1.570796, 1.671661],accel_mss,speed_ms,0,blend_radius_m)
    movel([0.101501, -1.480562, -2.488833, -0.742994, 1.570796, 1.672297],accel_mss,speed_ms,0,blend_radius_m)
    movel([0.102239, -1.480856, -2.488581, -0.742952, 1.570796, 1.673035],accel_mss,speed_ms,0,blend_radius_m)
    movel([0.103062, -1.481008, -2.488450, -0.742930, 1.570796, 1.673859],accel_mss,speed_ms,0,blend_radius_m)
    movel([0.103963, -1.481036, -2.488427, -0.742926, 1.570796, 1.674759],accel_mss,speed_ms,0,blend_radius_m)
    movel([0.104925, -1.480958, -2.488493, -0.742937, 1.570796, 1.675721],accel_mss,speed_ms,0,blend_radius_m)
    movel([0.108488, -1.480248, -2.489103, -0.743039, 1.570796, 1.679285],accel_mss,speed_ms,0,blend_radius_m)
    movel([0.108948, -1.480231, -2.489117, -0.743041, 1.570796, 1.679745],accel_mss,speed_ms,0,blend_radius_m)
    movel([0.109247, -1.480341, -2.489023, -0.743025, 1.570796, 1.680043],accel_mss,speed_ms,0,blend_radius_m)
    movel([0.109406, -1.480597, -2.488803, -0.742989, 1.570796, 1.680203],accel_mss,speed_ms,0,blend_radius_m)
    movel([0.109457, -1.481021, -2.488440, -0.742928, 1.570796, 1.680253],accel_mss,speed_ms,0,blend_radius_m)
    movel([0.109325, -1.482461, -2.487203, -0.742725, 1.570796, 1.680122],accel_mss,speed_ms,0,blend_radius_m)
    movel([0.107114, -1.483148, -2.486612, -0.742630, 1.570796, 1.677911],accel_mss,speed_ms,0,blend_radius_m)
    speed_ms = 0.005
    # Splitting Linear movement in 6 (instruction 99: MoveL 87)
    movel([0.107114, -1.481833, -2.486019, -0.744537, 1.570796, 1.677911],accel_mss,speed_ms,0,blend_radius_m)
    movel([0.107114, -1.480522, -2.485424, -0.746443, 1.570796, 1.677911],accel_mss,speed_ms,0,blend_radius_m)
    movel([0.107114, -1.479214, -2.484828, -0.748347, 1.570796, 1.677911],accel_mss,speed_ms,0,blend_radius_m)
    movel([0.107114, -1.477910, -2.484230, -0.750249, 1.570796, 1.677911],accel_mss,speed_ms,0,blend_radius_m)
    movel([0.107114, -1.476608, -2.483631, -0.752150, 1.570796, 1.677911],accel_mss,speed_ms,0,blend_radius_m)
    movel([0.107114, -1.475311, -2.483030, -0.754048, 1.570796, 1.677911],accel_mss,speed_ms,0,blend_radius_m)
    speed_ms = 0.040
    # Splitting Linear movement in 14 (instruction 101: MoveL 88)
    movel([0.106275, -1.473948, -2.484188, -0.754253, 1.570796, 1.677072],accel_mss,speed_ms,0,blend_radius_m)
    movel([0.105433, -1.472584, -2.485343, -0.754461, 1.570796, 1.676230],accel_mss,speed_ms,0,blend_radius_m)
    movel([0.104588, -1.471220, -2.486497, -0.754672, 1.570796, 1.675384],accel_mss,speed_ms,0,blend_radius_m)
    movel([0.103740, -1.469855, -2.487648, -0.754886, 1.570796, 1.674536],accel_mss,speed_ms,0,blend_radius_m)
    movel([0.102889, -1.468489, -2.488797, -0.755103, 1.570796, 1.673685],accel_mss,speed_ms,0,blend_radius_m)
    movel([0.102034, -1.467123, -2.489944, -0.755322, 1.570796, 1.672831],accel_mss,speed_ms,0,blend_radius_m)
    movel([0.101177, -1.465756, -2.491088, -0.755545, 1.570796, 1.671973],accel_mss,speed_ms,0,blend_radius_m)
    movel([0.100316, -1.464388, -2.492231, -0.755771, 1.570796, 1.671112],accel_mss,speed_ms,0,blend_radius_m)
    movel([0.099452, -1.463019, -2.493371, -0.756000, 1.570796, 1.670249],accel_mss,speed_ms,0,blend_radius_m)
    movel([0.098585, -1.461649, -2.494509, -0.756231, 1.570796, 1.669382],accel_mss,speed_ms,0,blend_radius_m)
    movel([0.097715, -1.460279, -2.495644, -0.756466, 1.570796, 1.668512],accel_mss,speed_ms,0,blend_radius_m)
    movel([0.096842, -1.458908, -2.496778, -0.756704, 1.570796, 1.667638],accel_mss,speed_ms,0,blend_radius_m)
    movel([0.095965, -1.457536, -2.497909, -0.756944, 1.570796, 1.666762],accel_mss,speed_ms,0,blend_radius_m)
    movel([0.095086, -1.456163, -2.499038, -0.757188, 1.570796, 1.665882],accel_mss,speed_ms,0,blend_radius_m)
    speed_ms = 0.005
    # Splitting Linear movement in 4 (instruction 103: MoveL 89)
    movel([0.095086, -1.458147, -2.499958, -0.754284, 1.570796, 1.665882],accel_mss,speed_ms,0,blend_radius_m)
    movel([0.095086, -1.460139, -2.500874, -0.751376, 1.570796, 1.665882],accel_mss,speed_ms,0,blend_radius_m)
    movel([0.095086, -1.462138, -2.501787, -0.748464, 1.570796, 1.665882],accel_mss,speed_ms,0,blend_radius_m)
    movel([0.095086, -1.464145, -2.502696, -0.745547, 1.570796, 1.665882],accel_mss,speed_ms,0,blend_radius_m)
    speed_ms = 0.035
    movel([0.094408, -1.462009, -2.504470, -0.745910, 1.570796, 1.665204],accel_mss,speed_ms,0,blend_radius_m)
    movel([0.097635, -1.459852, -2.506253, -0.746284, 1.570796, 1.668431],accel_mss,speed_ms,0,blend_radius_m)
    movel([0.098819, -1.458951, -2.506996, -0.746442, 1.570796, 1.669615],accel_mss,speed_ms,0,blend_radius_m)
    movel([0.099893, -1.458010, -2.507770, -0.746609, 1.570796, 1.670689],accel_mss,speed_ms,0,blend_radius_m)
    movel([0.100845, -1.457033, -2.508573, -0.746783, 1.570796, 1.671641],accel_mss,speed_ms,0,blend_radius_m)
    movel([0.101674, -1.456015, -2.509408, -0.746966, 1.570796, 1.672470],accel_mss,speed_ms,0,blend_radius_m)
    movel([0.102366, -1.454956, -2.510275, -0.747159, 1.570796, 1.673162],accel_mss,speed_ms,0,blend_radius_m)
    movel([0.102914, -1.453852, -2.511176, -0.747361, 1.570796, 1.673710],accel_mss,speed_ms,0,blend_radius_m)
    movel([0.103311, -1.452709, -2.512108, -0.747572, 1.570796, 1.674107],accel_mss,speed_ms,0,blend_radius_m)
    movel([0.103546, -1.451519, -2.513075, -0.747794, 1.570796, 1.674342],accel_mss,speed_ms,0,blend_radius_m)
    movel([0.103749, -1.450763, -2.513689, -0.747937, 1.570796, 1.674545],accel_mss,speed_ms,0,blend_radius_m)
    movel([0.104143, -1.450242, -2.514112, -0.748035, 1.570796, 1.674939],accel_mss,speed_ms,0,blend_radius_m)
    movel([0.104744, -1.449884, -2.514401, -0.748103, 1.570796, 1.675540],accel_mss,speed_ms,0,blend_radius_m)
    movel([0.105564, -1.449622, -2.514614, -0.748153, 1.570796, 1.676361],accel_mss,speed_ms,0,blend_radius_m)
    movel([0.106357, -1.449514, -2.514701, -0.748174, 1.570796, 1.677153],accel_mss,speed_ms,0,blend_radius_m)
    movel([0.106803, -1.449677, -2.514570, -0.748143, 1.570796, 1.677599],accel_mss,speed_ms,0,blend_radius_m)
    movel([0.106975, -1.450088, -2.514236, -0.748064, 1.570796, 1.677772],accel_mss,speed_ms,0,blend_radius_m)
    movel([0.106958, -1.450724, -2.513721, -0.747944, 1.570796, 1.677754],accel_mss,speed_ms,0,blend_radius_m)
    movel([0.106539, -1.452607, -2.512191, -0.747591, 1.570796, 1.677335],accel_mss,speed_ms,0,blend_radius_m)
    movel([0.105755, -1.454506, -2.510643, -0.747241, 1.570796, 1.676551],accel_mss,speed_ms,0,blend_radius_m)
    movel([0.104635, -1.456382, -2.509107, -0.746900, 1.570796, 1.675431],accel_mss,speed_ms,0,blend_radius_m)
    movel([0.103212, -1.458196, -2.507617, -0.746576, 1.570796, 1.674008],accel_mss,speed_ms,0,blend_radius_m)
    movel([0.101515, -1.459917, -2.506199, -0.746273, 1.570796, 1.672311],accel_mss,speed_ms,0,blend_radius_m)
    movel([0.099576, -1.461503, -2.504888, -0.745997, 1.570796, 1.670372],accel_mss,speed_ms,0,blend_radius_m)
    movel([0.097423, -1.462925, -2.503710, -0.745754, 1.570796, 1.668219],accel_mss,speed_ms,0,blend_radius_m)
    movel([0.095086, -1.464145, -2.502696, -0.745547, 1.570796, 1.665882],accel_mss,speed_ms,0,blend_radius_m)
    movel([0.094565, -1.462505, -2.504059, -0.745826, 1.570796, 1.665362],accel_mss,speed_ms,0,blend_radius_m)
    speed_ms = 0.005
    # Splitting Linear movement in 4 (instruction 133: MoveL 117)
    movel([0.094565, -1.460494, -2.503148, -0.748747, 1.570796, 1.665362],accel_mss,speed_ms,0,blend_radius_m)
    movel([0.094565, -1.458492, -2.502233, -0.751664, 1.570796, 1.665362],accel_mss,speed_ms,0,blend_radius_m)
    movel([0.094565, -1.456497, -2.501315, -0.754577, 1.570796, 1.665362],accel_mss,speed_ms,0,blend_radius_m)
    movel([0.094565, -1.454510, -2.500394, -0.757485, 1.570796, 1.665362],accel_mss,speed_ms,0,blend_radius_m)
    speed_ms = 0.040
    # Splitting Linear movement in 18 (instruction 135: MoveL 118)
    movel([0.094508, -1.452787, -2.501803, -0.757799, 1.570796, 1.665304],accel_mss,speed_ms,0,blend_radius_m)
    movel([0.094450, -1.451060, -2.503210, -0.758119, 1.570796, 1.665246],accel_mss,speed_ms,0,blend_radius_m)
    movel([0.094391, -1.449329, -2.504616, -0.758444, 1.570796, 1.665188],accel_mss,speed_ms,0,blend_radius_m)
    movel([0.094333, -1.447594, -2.506021, -0.758773, 1.570796, 1.665129],accel_mss,speed_ms,0,blend_radius_m)
    movel([0.094274, -1.445856, -2.507425, -0.759109, 1.570796, 1.665071],accel_mss,speed_ms,0,blend_radius_m)
    movel([0.094215, -1.444113, -2.508826, -0.759449, 1.570796, 1.665012],accel_mss,speed_ms,0,blend_radius_m)
    movel([0.094156, -1.442367, -2.510227, -0.759795, 1.570796, 1.664952],accel_mss,speed_ms,0,blend_radius_m)
    movel([0.094097, -1.440617, -2.511626, -0.760146, 1.570796, 1.664893],accel_mss,speed_ms,0,blend_radius_m)
    movel([0.094037, -1.438863, -2.513023, -0.760503, 1.570796, 1.664833],accel_mss,speed_ms,0,blend_radius_m)
    movel([0.093977, -1.437105, -2.514419, -0.760865, 1.570796, 1.664773],accel_mss,speed_ms,0,blend_radius_m)
    movel([0.093917, -1.435343, -2.515814, -0.761233, 1.570796, 1.664713],accel_mss,speed_ms,0,blend_radius_m)
    movel([0.093856, -1.433577, -2.517207, -0.761606, 1.570796, 1.664653],accel_mss,speed_ms,0,blend_radius_m)
    movel([0.093796, -1.431807, -2.518598, -0.761984, 1.570796, 1.664592],accel_mss,speed_ms,0,blend_radius_m)
    movel([0.093735, -1.430033, -2.519988, -0.762368, 1.570796, 1.664531],accel_mss,speed_ms,0,blend_radius_m)
    movel([0.093673, -1.428254, -2.521377, -0.762758, 1.570796, 1.664470],accel_mss,speed_ms,0,blend_radius_m)
    movel([0.093612, -1.426472, -2.522764, -0.763153, 1.570796, 1.664408],accel_mss,speed_ms,0,blend_radius_m)
    movel([0.093550, -1.424686, -2.524149, -0.763554, 1.570796, 1.664346],accel_mss,speed_ms,0,blend_radius_m)
    movel([0.093488, -1.422895, -2.525533, -0.763961, 1.570796, 1.664284],accel_mss,speed_ms,0,blend_radius_m)
    speed_ms = 0.005
    # Splitting Linear movement in 6 (instruction 137: MoveL 119)
    movel([0.093488, -1.424257, -2.526169, -0.761962, 1.570796, 1.664284],accel_mss,speed_ms,0,blend_radius_m)
    movel([0.093488, -1.425623, -2.526804, -0.759962, 1.570796, 1.664284],accel_mss,speed_ms,0,blend_radius_m)
    movel([0.093488, -1.426993, -2.527438, -0.757959, 1.570796, 1.664284],accel_mss,speed_ms,0,blend_radius_m)
    movel([0.093488, -1.428366, -2.528069, -0.755954, 1.570796, 1.664284],accel_mss,speed_ms,0,blend_radius_m)
    movel([0.093488, -1.429743, -2.528699, -0.753946, 1.570796, 1.664284],accel_mss,speed_ms,0,blend_radius_m)
    movel([0.093488, -1.431124, -2.529328, -0.751937, 1.570796, 1.664284],accel_mss,speed_ms,0,blend_radius_m)
    speed_ms = 0.035
    # Splitting Linear movement in 4 (instruction 139: MoveL 120)
    movel([0.095293, -1.430651, -2.529698, -0.752041, 1.570796, 1.666089],accel_mss,speed_ms,0,blend_radius_m)
    movel([0.097098, -1.430179, -2.530066, -0.752144, 1.570796, 1.667895],accel_mss,speed_ms,0,blend_radius_m)
    movel([0.098905, -1.429710, -2.530431, -0.752248, 1.570796, 1.669701],accel_mss,speed_ms,0,blend_radius_m)
    movel([0.100712, -1.429243, -2.530795, -0.752351, 1.570796, 1.671508],accel_mss,speed_ms,0,blend_radius_m)
    movel([0.101513, -1.429109, -2.530900, -0.752381, 1.570796, 1.672310],accel_mss,speed_ms,0,blend_radius_m)
    movel([0.102000, -1.429245, -2.530794, -0.752350, 1.570796, 1.672796],accel_mss,speed_ms,0,blend_radius_m)
    movel([0.102216, -1.429647, -2.530480, -0.752261, 1.570796, 1.673012],accel_mss,speed_ms,0,blend_radius_m)
    movel([0.102214, -1.430310, -2.529964, -0.752115, 1.570796, 1.673011],accel_mss,speed_ms,0,blend_radius_m)
    movel([0.102036, -1.431025, -2.529406, -0.751959, 1.570796, 1.672832],accel_mss,speed_ms,0,blend_radius_m)
    movel([0.101677, -1.431556, -2.528990, -0.751843, 1.570796, 1.672474],accel_mss,speed_ms,0,blend_radius_m)
    movel([0.101110, -1.431940, -2.528690, -0.751759, 1.570796, 1.671906],accel_mss,speed_ms,0,blend_radius_m)
    movel([0.100306, -1.432214, -2.528475, -0.751700, 1.570796, 1.671102],accel_mss,speed_ms,0,blend_radius_m)
    # Splitting Linear movement in 8 (instruction 148: MoveL 129)
    movel([0.098506, -1.432671, -2.528117, -0.751601, 1.570796, 1.669303],accel_mss,speed_ms,0,blend_radius_m)
    movel([0.096708, -1.433130, -2.527758, -0.751502, 1.570796, 1.667504],accel_mss,speed_ms,0,blend_radius_m)
    movel([0.094909, -1.433590, -2.527396, -0.751403, 1.570796, 1.665706],accel_mss,speed_ms,0,blend_radius_m)
    movel([0.093112, -1.434054, -2.527032, -0.751303, 1.570796, 1.663908],accel_mss,speed_ms,0,blend_radius_m)
    movel([0.091315, -1.434519, -2.526666, -0.751204, 1.570796, 1.662111],accel_mss,speed_ms,0,blend_radius_m)
    movel([0.089519, -1.434986, -2.526299, -0.751104, 1.570796, 1.660315],accel_mss,speed_ms,0,blend_radius_m)
    movel([0.087724, -1.435455, -2.525929, -0.751005, 1.570796, 1.658520],accel_mss,speed_ms,0,blend_radius_m)
    movel([0.085929, -1.435927, -2.525557, -0.750905, 1.570796, 1.656725],accel_mss,speed_ms,0,blend_radius_m)
    movel([0.085098, -1.436068, -2.525446, -0.750875, 1.570796, 1.655894],accel_mss,speed_ms,0,blend_radius_m)
    movel([0.084565, -1.435948, -2.525540, -0.750900, 1.570796, 1.655361],accel_mss,speed_ms,0,blend_radius_m)
    movel([0.084301, -1.435545, -2.525859, -0.750986, 1.570796, 1.655097],accel_mss,speed_ms,0,blend_radius_m)
    movel([0.084287, -1.434834, -2.526419, -0.751137, 1.570796, 1.655084],accel_mss,speed_ms,0,blend_radius_m)
    movel([0.084500, -1.434085, -2.527008, -0.751297, 1.570796, 1.655297],accel_mss,speed_ms,0,blend_radius_m)
    movel([0.084917, -1.433580, -2.527404, -0.751405, 1.570796, 1.655713],accel_mss,speed_ms,0,blend_radius_m)
    movel([0.085517, -1.433249, -2.527664, -0.751476, 1.570796, 1.656313],accel_mss,speed_ms,0,blend_radius_m)
    movel([0.086281, -1.433013, -2.527849, -0.751527, 1.570796, 1.657077],accel_mss,speed_ms,0,blend_radius_m)
    # Splitting Linear movement in 4 (instruction 157: MoveL 138)
    movel([0.088081, -1.432538, -2.528222, -0.751630, 1.570796, 1.658878],accel_mss,speed_ms,0,blend_radius_m)
    movel([0.089883, -1.432064, -2.528592, -0.751732, 1.570796, 1.660679],accel_mss,speed_ms,0,blend_radius_m)
    movel([0.091685, -1.431593, -2.528961, -0.751835, 1.570796, 1.662481],accel_mss,speed_ms,0,blend_radius_m)
    movel([0.093488, -1.431124, -2.529328, -0.751937, 1.570796, 1.664284],accel_mss,speed_ms,0,blend_radius_m)
    movel([0.095833, -1.430509, -2.529808, -0.752072, 1.570796, 1.666629],accel_mss,speed_ms,0,blend_radius_m)
    speed_ms = 0.005
    # Splitting Linear movement in 6 (instruction 160: MoveL 140)
    movel([0.095833, -1.429127, -2.529179, -0.754082, 1.570796, 1.666629],accel_mss,speed_ms,0,blend_radius_m)
    movel([0.095833, -1.427749, -2.528549, -0.756091, 1.570796, 1.666629],accel_mss,speed_ms,0,blend_radius_m)
    movel([0.095833, -1.426375, -2.527917, -0.758097, 1.570796, 1.666629],accel_mss,speed_ms,0,blend_radius_m)
    movel([0.095833, -1.425005, -2.527283, -0.760101, 1.570796, 1.666629],accel_mss,speed_ms,0,blend_radius_m)
    movel([0.095833, -1.423639, -2.526648, -0.762103, 1.570796, 1.666629],accel_mss,speed_ms,0,blend_radius_m)
    movel([0.095833, -1.422276, -2.526011, -0.764102, 1.570796, 1.666629],accel_mss,speed_ms,0,blend_radius_m)
    speed_ms = 0.040
    # Splitting Linear movement in 16 (instruction 162: MoveL 141)
    movel([0.097717, -1.420624, -2.527282, -0.764483, 1.570796, 1.668513],accel_mss,speed_ms,0,blend_radius_m)
    movel([0.099607, -1.418969, -2.528551, -0.764869, 1.570796, 1.670403],accel_mss,speed_ms,0,blend_radius_m)
    movel([0.101503, -1.417311, -2.529819, -0.765259, 1.570796, 1.672299],accel_mss,speed_ms,0,blend_radius_m)
    movel([0.103405, -1.415650, -2.531084, -0.765654, 1.570796, 1.674201],accel_mss,speed_ms,0,blend_radius_m)
    movel([0.105313, -1.413987, -2.532348, -0.766054, 1.570796, 1.676110],accel_mss,speed_ms,0,blend_radius_m)
    movel([0.107228, -1.412321, -2.533610, -0.766458, 1.570796, 1.678024],accel_mss,speed_ms,0,blend_radius_m)
    movel([0.109148, -1.410652, -2.534869, -0.766868, 1.570796, 1.679945],accel_mss,speed_ms,0,blend_radius_m)
    movel([0.111075, -1.408980, -2.536127, -0.767281, 1.570796, 1.681872],accel_mss,speed_ms,0,blend_radius_m)
    movel([0.113008, -1.407306, -2.537383, -0.767700, 1.570796, 1.683805],accel_mss,speed_ms,0,blend_radius_m)
    movel([0.114947, -1.405628, -2.538637, -0.768124, 1.570796, 1.685744],accel_mss,speed_ms,0,blend_radius_m)
    movel([0.116893, -1.403948, -2.539888, -0.768552, 1.570796, 1.687689],accel_mss,speed_ms,0,blend_radius_m)
    movel([0.118845, -1.402265, -2.541138, -0.768985, 1.570796, 1.689641],accel_mss,speed_ms,0,blend_radius_m)
    movel([0.120803, -1.400579, -2.542386, -0.769423, 1.570796, 1.691599],accel_mss,speed_ms,0,blend_radius_m)
    movel([0.122767, -1.398891, -2.543632, -0.769866, 1.570796, 1.693563],accel_mss,speed_ms,0,blend_radius_m)
    movel([0.124738, -1.397199, -2.544876, -0.770314, 1.570796, 1.695534],accel_mss,speed_ms,0,blend_radius_m)
    movel([0.126715, -1.395505, -2.546117, -0.770767, 1.570796, 1.697511],accel_mss,speed_ms,0,blend_radius_m)
    speed_ms = 0.005
    # Splitting Linear movement in 4 (instruction 164: MoveL 142)
    movel([0.126715, -1.397597, -2.547100, -0.767691, 1.570796, 1.697511],accel_mss,speed_ms,0,blend_radius_m)
    movel([0.126715, -1.399699, -2.548080, -0.764610, 1.570796, 1.697511],accel_mss,speed_ms,0,blend_radius_m)
    movel([0.126715, -1.401810, -2.549056, -0.761524, 1.570796, 1.697511],accel_mss,speed_ms,0,blend_radius_m)
    movel([0.126715, -1.403930, -2.550028, -0.758432, 1.570796, 1.697511],accel_mss,speed_ms,0,blend_radius_m)
    speed_ms = 0.035
    # Splitting Linear movement in 4 (instruction 166: MoveL 143)
    movel([0.127916, -1.404166, -2.549852, -0.758370, 1.570796, 1.698712],accel_mss,speed_ms,0,blend_radius_m)
    movel([0.129116, -1.404404, -2.549676, -0.758309, 1.570796, 1.699912],accel_mss,speed_ms,0,blend_radius_m)
    movel([0.130314, -1.404644, -2.549498, -0.758247, 1.570796, 1.701111],accel_mss,speed_ms,0,blend_radius_m)
    movel([0.131512, -1.404885, -2.549319, -0.758185, 1.570796, 1.702308],accel_mss,speed_ms,0,blend_radius_m)
    # Splitting Linear movement in 10 (instruction 167: MoveL 144)
    movel([0.133306, -1.405261, -2.549040, -0.758088, 1.570796, 1.704102],accel_mss,speed_ms,0,blend_radius_m)
    movel([0.135097, -1.405640, -2.548758, -0.757991, 1.570796, 1.705893],accel_mss,speed_ms,0,blend_radius_m)
    movel([0.136885, -1.406023, -2.548473, -0.757893, 1.570796, 1.707681],accel_mss,speed_ms,0,blend_radius_m)
    movel([0.138670, -1.406410, -2.548185, -0.757794, 1.570796, 1.709467],accel_mss,speed_ms,0,blend_radius_m)
    movel([0.140452, -1.406799, -2.547895, -0.757695, 1.570796, 1.711249],accel_mss,speed_ms,0,blend_radius_m)
    movel([0.142231, -1.407193, -2.547602, -0.757594, 1.570796, 1.713028],accel_mss,speed_ms,0,blend_radius_m)
    movel([0.144008, -1.407590, -2.547306, -0.757494, 1.570796, 1.714804],accel_mss,speed_ms,0,blend_radius_m)
    movel([0.145781, -1.407990, -2.547007, -0.757392, 1.570796, 1.716577],accel_mss,speed_ms,0,blend_radius_m)
    movel([0.147551, -1.408394, -2.546705, -0.757290, 1.570796, 1.718347],accel_mss,speed_ms,0,blend_radius_m)
    movel([0.149318, -1.408801, -2.546400, -0.757188, 1.570796, 1.720114],accel_mss,speed_ms,0,blend_radius_m)
    movel([0.150561, -1.409178, -2.546118, -0.757093, 1.570796, 1.721357],accel_mss,speed_ms,0,blend_radius_m)
    movel([0.151594, -1.409751, -2.545689, -0.756949, 1.570796, 1.722391],accel_mss,speed_ms,0,blend_radius_m)
    movel([0.152000, -1.410136, -2.545400, -0.756853, 1.570796, 1.722797],accel_mss,speed_ms,0,blend_radius_m)
    movel([0.152314, -1.410600, -2.545052, -0.756737, 1.570796, 1.723110],accel_mss,speed_ms,0,blend_radius_m)
    movel([0.152520, -1.411154, -2.544636, -0.756599, 1.570796, 1.723316],accel_mss,speed_ms,0,blend_radius_m)
    movel([0.152610, -1.411807, -2.544144, -0.756437, 1.570796, 1.723406],accel_mss,speed_ms,0,blend_radius_m)
    movel([0.152506, -1.412845, -2.543363, -0.756182, 1.570796, 1.723302],accel_mss,speed_ms,0,blend_radius_m)
    movel([0.152142, -1.413882, -2.542580, -0.755928, 1.570796, 1.722939],accel_mss,speed_ms,0,blend_radius_m)
    movel([0.151550, -1.414883, -2.541822, -0.755684, 1.570796, 1.722346],accel_mss,speed_ms,0,blend_radius_m)
    movel([0.150755, -1.415823, -2.541110, -0.755456, 1.570796, 1.721551],accel_mss,speed_ms,0,blend_radius_m)
    movel([0.149785, -1.416675, -2.540463, -0.755251, 1.570796, 1.720581],accel_mss,speed_ms,0,blend_radius_m)
    movel([0.148671, -1.417406, -2.539907, -0.755076, 1.570796, 1.719467],accel_mss,speed_ms,0,blend_radius_m)
    movel([0.147440, -1.417990, -2.539463, -0.754937, 1.570796, 1.718236],accel_mss,speed_ms,0,blend_radius_m)
    movel([0.146116, -1.418399, -2.539151, -0.754839, 1.570796, 1.716912],accel_mss,speed_ms,0,blend_radius_m)
    # Splitting Linear movement in 8 (instruction 182: MoveL 159)
    movel([0.143924, -1.418886, -2.538779, -0.754724, 1.570796, 1.714720],accel_mss,speed_ms,0,blend_radius_m)
    movel([0.141732, -1.419377, -2.538404, -0.754608, 1.570796, 1.712528],accel_mss,speed_ms,0,blend_radius_m)
    movel([0.139541, -1.419871, -2.538027, -0.754491, 1.570796, 1.710337],accel_mss,speed_ms,0,blend_radius_m)
    movel([0.137350, -1.420369, -2.537646, -0.754374, 1.570796, 1.708146],accel_mss,speed_ms,0,blend_radius_m)
    movel([0.135160, -1.420870, -2.537263, -0.754257, 1.570796, 1.705956],accel_mss,speed_ms,0,blend_radius_m)
    movel([0.132971, -1.421374, -2.536876, -0.754139, 1.570796, 1.703767],accel_mss,speed_ms,0,blend_radius_m)
    movel([0.130782, -1.421882, -2.536486, -0.754021, 1.570796, 1.701579],accel_mss,speed_ms,0,blend_radius_m)
    movel([0.128595, -1.422393, -2.536094, -0.753902, 1.570796, 1.699391],accel_mss,speed_ms,0,blend_radius_m)
    movel([0.127707, -1.422683, -2.535871, -0.753835, 1.570796, 1.698503],accel_mss,speed_ms,0,blend_radius_m)
    movel([0.127123, -1.423091, -2.535557, -0.753741, 1.570796, 1.697919],accel_mss,speed_ms,0,blend_radius_m)
    movel([0.126772, -1.423657, -2.535121, -0.753611, 1.570796, 1.697568],accel_mss,speed_ms,0,blend_radius_m)
    movel([0.126581, -1.424410, -2.534540, -0.753438, 1.570796, 1.697378],accel_mss,speed_ms,0,blend_radius_m)
    movel([0.126552, -1.424861, -2.534192, -0.753335, 1.570796, 1.697348],accel_mss,speed_ms,0,blend_radius_m)
    movel([0.126785, -1.425378, -2.533793, -0.753218, 1.570796, 1.697581],accel_mss,speed_ms,0,blend_radius_m)
    movel([0.127017, -1.425483, -2.533712, -0.753194, 1.570796, 1.697813],accel_mss,speed_ms,0,blend_radius_m)
    movel([0.127657, -1.425479, -2.533716, -0.753195, 1.570796, 1.698454],accel_mss,speed_ms,0,blend_radius_m)
    movel([0.128440, -1.425313, -2.533844, -0.753232, 1.570796, 1.699236],accel_mss,speed_ms,0,blend_radius_m)
    # Splitting Linear movement in 8 (instruction 192: MoveL 169)
    movel([0.130720, -1.424769, -2.534264, -0.753356, 1.570796, 1.701517],accel_mss,speed_ms,0,blend_radius_m)
    movel([0.133001, -1.424228, -2.534681, -0.753480, 1.570796, 1.703798],accel_mss,speed_ms,0,blend_radius_m)
    movel([0.135283, -1.423690, -2.535096, -0.753603, 1.570796, 1.706080],accel_mss,speed_ms,0,blend_radius_m)
    movel([0.137566, -1.423157, -2.535506, -0.753726, 1.570796, 1.708362],accel_mss,speed_ms,0,blend_radius_m)
    movel([0.139850, -1.422627, -2.535914, -0.753848, 1.570796, 1.710646],accel_mss,speed_ms,0,blend_radius_m)
    movel([0.142134, -1.422100, -2.536318, -0.753970, 1.570796, 1.712930],accel_mss,speed_ms,0,blend_radius_m)
    movel([0.144419, -1.421578, -2.536720, -0.754092, 1.570796, 1.715215],accel_mss,speed_ms,0,blend_radius_m)
    movel([0.146705, -1.421059, -2.537118, -0.754213, 1.570796, 1.717501],accel_mss,speed_ms,0,blend_radius_m)
    movel([0.147624, -1.420791, -2.537323, -0.754275, 1.570796, 1.718420],accel_mss,speed_ms,0,blend_radius_m)
    movel([0.149504, -1.419967, -2.537954, -0.754469, 1.570796, 1.720300],accel_mss,speed_ms,0,blend_radius_m)
    movel([0.150393, -1.419446, -2.538352, -0.754591, 1.570796, 1.721189],accel_mss,speed_ms,0,blend_radius_m)
    movel([0.151559, -1.418629, -2.538975, -0.754785, 1.570796, 1.722356],accel_mss,speed_ms,0,blend_radius_m)
    movel([0.152591, -1.417758, -2.539639, -0.754992, 1.570796, 1.723388],accel_mss,speed_ms,0,blend_radius_m)
    movel([0.153490, -1.416837, -2.540340, -0.755212, 1.570796, 1.724287],accel_mss,speed_ms,0,blend_radius_m)
    movel([0.154255, -1.415870, -2.541074, -0.755445, 1.570796, 1.725052],accel_mss,speed_ms,0,blend_radius_m)
    movel([0.154893, -1.414859, -2.541840, -0.755689, 1.570796, 1.725689],accel_mss,speed_ms,0,blend_radius_m)
    movel([0.155401, -1.413809, -2.542635, -0.755945, 1.570796, 1.726197],accel_mss,speed_ms,0,blend_radius_m)
    movel([0.155784, -1.412724, -2.543454, -0.756211, 1.570796, 1.726580],accel_mss,speed_ms,0,blend_radius_m)
    movel([0.156043, -1.411604, -2.544297, -0.756488, 1.570796, 1.726840],accel_mss,speed_ms,0,blend_radius_m)
    movel([0.156154, -1.410494, -2.545131, -0.756764, 1.570796, 1.726951],accel_mss,speed_ms,0,blend_radius_m)
    movel([0.156082, -1.409501, -2.545876, -0.757012, 1.570796, 1.726878],accel_mss,speed_ms,0,blend_radius_m)
    movel([0.155834, -1.408626, -2.546531, -0.757232, 1.570796, 1.726630],accel_mss,speed_ms,0,blend_radius_m)
    movel([0.155422, -1.407868, -2.547098, -0.757423, 1.570796, 1.726218],accel_mss,speed_ms,0,blend_radius_m)
    movel([0.154853, -1.407222, -2.547580, -0.757587, 1.570796, 1.725650],accel_mss,speed_ms,0,blend_radius_m)
    movel([0.154139, -1.406692, -2.547975, -0.757722, 1.570796, 1.724936],accel_mss,speed_ms,0,blend_radius_m)
    movel([0.153287, -1.406271, -2.548289, -0.757829, 1.570796, 1.724083],accel_mss,speed_ms,0,blend_radius_m)
    movel([0.152307, -1.405959, -2.548521, -0.757909, 1.570796, 1.723103],accel_mss,speed_ms,0,blend_radius_m)
    # Splitting Linear movement in 14 (instruction 212: MoveL 189)
    movel([0.150360, -1.405502, -2.548861, -0.758026, 1.570796, 1.721157],accel_mss,speed_ms,0,blend_radius_m)
    movel([0.148410, -1.405048, -2.549198, -0.758143, 1.570796, 1.719206],accel_mss,speed_ms,0,blend_radius_m)
    movel([0.146456, -1.404600, -2.549531, -0.758258, 1.570796, 1.717252],accel_mss,speed_ms,0,blend_radius_m)
    movel([0.144498, -1.404155, -2.549861, -0.758373, 1.570796, 1.715294],accel_mss,speed_ms,0,blend_radius_m)
    movel([0.142537, -1.403714, -2.550187, -0.758487, 1.570796, 1.713333],accel_mss,speed_ms,0,blend_radius_m)
    movel([0.140571, -1.403278, -2.550510, -0.758601, 1.570796, 1.711368],accel_mss,speed_ms,0,blend_radius_m)
    movel([0.138603, -1.402846, -2.550830, -0.758713, 1.570796, 1.709399],accel_mss,speed_ms,0,blend_radius_m)
    movel([0.136630, -1.402419, -2.551146, -0.758825, 1.570796, 1.707426],accel_mss,speed_ms,0,blend_radius_m)
    movel([0.134654, -1.401995, -2.551459, -0.758935, 1.570796, 1.705450],accel_mss,speed_ms,0,blend_radius_m)
    movel([0.132674, -1.401576, -2.551768, -0.759045, 1.570796, 1.703470],accel_mss,speed_ms,0,blend_radius_m)
    movel([0.130690, -1.401161, -2.552074, -0.759154, 1.570796, 1.701486],accel_mss,speed_ms,0,blend_radius_m)
    movel([0.128703, -1.400751, -2.552376, -0.759262, 1.570796, 1.699499],accel_mss,speed_ms,0,blend_radius_m)
    movel([0.126712, -1.400344, -2.552675, -0.759369, 1.570796, 1.697508],accel_mss,speed_ms,0,blend_radius_m)
    movel([0.124717, -1.399942, -2.552971, -0.759476, 1.570796, 1.695514],accel_mss,speed_ms,0,blend_radius_m)
    movel([0.123823, -1.400080, -2.552870, -0.759439, 1.570796, 1.694619],accel_mss,speed_ms,0,blend_radius_m)
    # Splitting Linear movement in 16 (instruction 214: MoveL 191)
    movel([0.123525, -1.402154, -2.551342, -0.758894, 1.570796, 1.694321],accel_mss,speed_ms,0,blend_radius_m)
    movel([0.123228, -1.404221, -2.549812, -0.758356, 1.570796, 1.694025],accel_mss,speed_ms,0,blend_radius_m)
    movel([0.122933, -1.406282, -2.548280, -0.757826, 1.570796, 1.693729],accel_mss,speed_ms,0,blend_radius_m)
    movel([0.122639, -1.408338, -2.546747, -0.757305, 1.570796, 1.693436],accel_mss,speed_ms,0,blend_radius_m)
    movel([0.122347, -1.410386, -2.545212, -0.756790, 1.570796, 1.693143],accel_mss,speed_ms,0,blend_radius_m)
    movel([0.122056, -1.412429, -2.543676, -0.756284, 1.570796, 1.692852],accel_mss,speed_ms,0,blend_radius_m)
    movel([0.121766, -1.414466, -2.542138, -0.755785, 1.570796, 1.692563],accel_mss,speed_ms,0,blend_radius_m)
    movel([0.121478, -1.416496, -2.540599, -0.755294, 1.570796, 1.692275],accel_mss,speed_ms,0,blend_radius_m)
    movel([0.121191, -1.418521, -2.539058, -0.754810, 1.570796, 1.691988],accel_mss,speed_ms,0,blend_radius_m)
    movel([0.120906, -1.420540, -2.537515, -0.754334, 1.570796, 1.691702],accel_mss,speed_ms,0,blend_radius_m)
    movel([0.120622, -1.422552, -2.535971, -0.753865, 1.570796, 1.691418],accel_mss,speed_ms,0,blend_radius_m)
    movel([0.120339, -1.424559, -2.534426, -0.753404, 1.570796, 1.691136],accel_mss,speed_ms,0,blend_radius_m)
    movel([0.120058, -1.426560, -2.532879, -0.752950, 1.570796, 1.690854],accel_mss,speed_ms,0,blend_radius_m)
    movel([0.119778, -1.428555, -2.531330, -0.752503, 1.570796, 1.690574],accel_mss,speed_ms,0,blend_radius_m)
    movel([0.119499, -1.430545, -2.529780, -0.752064, 1.570796, 1.690295],accel_mss,speed_ms,0,blend_radius_m)
    movel([0.119222, -1.432528, -2.528229, -0.751632, 1.570796, 1.690018],accel_mss,speed_ms,0,blend_radius_m)
    movel([0.119226, -1.433422, -2.527528, -0.751439, 1.570796, 1.690023],accel_mss,speed_ms,0,blend_radius_m)
    movel([0.119359, -1.433687, -2.527320, -0.751382, 1.570796, 1.690155],accel_mss,speed_ms,0,blend_radius_m)
    movel([0.119573, -1.433846, -2.527195, -0.751348, 1.570796, 1.690369],accel_mss,speed_ms,0,blend_radius_m)
    movel([0.120234, -1.433903, -2.527150, -0.751336, 1.570796, 1.691030],accel_mss,speed_ms,0,blend_radius_m)
    movel([0.121194, -1.433690, -2.527318, -0.751381, 1.570796, 1.691990],accel_mss,speed_ms,0,blend_radius_m)
    movel([0.121707, -1.433500, -2.527467, -0.751422, 1.570796, 1.692504],accel_mss,speed_ms,0,blend_radius_m)
    movel([0.122081, -1.433275, -2.527643, -0.751470, 1.570796, 1.692878],accel_mss,speed_ms,0,blend_radius_m)
    movel([0.122340, -1.433021, -2.527842, -0.751525, 1.570796, 1.693137],accel_mss,speed_ms,0,blend_radius_m)
    movel([0.122506, -1.432747, -2.528058, -0.751584, 1.570796, 1.693302],accel_mss,speed_ms,0,blend_radius_m)
    movel([0.122653, -1.432154, -2.528522, -0.751713, 1.570796, 1.693450],accel_mss,speed_ms,0,blend_radius_m)
    movel([0.122716, -1.431555, -2.528991, -0.751843, 1.570796, 1.693512],accel_mss,speed_ms,0,blend_radius_m)
    # Splitting Linear movement in 14 (instruction 226: MoveL 203)
    movel([0.122993, -1.429618, -2.530503, -0.752268, 1.570796, 1.693789],accel_mss,speed_ms,0,blend_radius_m)
    movel([0.123271, -1.427676, -2.532013, -0.752700, 1.570796, 1.694068],accel_mss,speed_ms,0,blend_radius_m)
    movel([0.123551, -1.425728, -2.533523, -0.753138, 1.570796, 1.694347],accel_mss,speed_ms,0,blend_radius_m)
    movel([0.123832, -1.423775, -2.535030, -0.753584, 1.570796, 1.694628],accel_mss,speed_ms,0,blend_radius_m)
    movel([0.124114, -1.421816, -2.536537, -0.754036, 1.570796, 1.694911],accel_mss,speed_ms,0,blend_radius_m)
    movel([0.124398, -1.419852, -2.538041, -0.754496, 1.570796, 1.695194],accel_mss,speed_ms,0,blend_radius_m)
    movel([0.124683, -1.417882, -2.539545, -0.754962, 1.570796, 1.695479],accel_mss,speed_ms,0,blend_radius_m)
    movel([0.124969, -1.415906, -2.541047, -0.755436, 1.570796, 1.695765],accel_mss,speed_ms,0,blend_radius_m)
    movel([0.125257, -1.413925, -2.542547, -0.755917, 1.570796, 1.696053],accel_mss,speed_ms,0,blend_radius_m)
    movel([0.125546, -1.411937, -2.544046, -0.756405, 1.570796, 1.696342],accel_mss,speed_ms,0,blend_radius_m)
    movel([0.125836, -1.409944, -2.545544, -0.756901, 1.570796, 1.696632],accel_mss,speed_ms,0,blend_radius_m)
    movel([0.126128, -1.407946, -2.547040, -0.757404, 1.570796, 1.696924],accel_mss,speed_ms,0,blend_radius_m)
    movel([0.126421, -1.405941, -2.548534, -0.757914, 1.570796, 1.697217],accel_mss,speed_ms,0,blend_radius_m)
    movel([0.126715, -1.403930, -2.550028, -0.758432, 1.570796, 1.697511],accel_mss,speed_ms,0,blend_radius_m)
    movel([0.128744, -1.404331, -2.549730, -0.758328, 1.570796, 1.699541],accel_mss,speed_ms,0,blend_radius_m)
    speed_ms = 0.005
    # Splitting Linear movement in 6 (instruction 229: MoveL 205)
    movel([0.128744, -1.402917, -2.549083, -0.760389, 1.570796, 1.699541],accel_mss,speed_ms,0,blend_radius_m)
    movel([0.128744, -1.401507, -2.548434, -0.762448, 1.570796, 1.699541],accel_mss,speed_ms,0,blend_radius_m)
    movel([0.128744, -1.400101, -2.547783, -0.764504, 1.570796, 1.699541],accel_mss,speed_ms,0,blend_radius_m)
    movel([0.128744, -1.398700, -2.547131, -0.766558, 1.570796, 1.699541],accel_mss,speed_ms,0,blend_radius_m)
    movel([0.128744, -1.397302, -2.546477, -0.768610, 1.570796, 1.699541],accel_mss,speed_ms,0,blend_radius_m)
    movel([0.128744, -1.395909, -2.545822, -0.770659, 1.570796, 1.699541],accel_mss,speed_ms,0,blend_radius_m)
    speed_ms = 0.040
    # Splitting Linear movement in 12 (instruction 231: MoveL 206)
    movel([0.127186, -1.395262, -2.546295, -0.770832, 1.570796, 1.697982],accel_mss,speed_ms,0,blend_radius_m)
    movel([0.125624, -1.394619, -2.546765, -0.771005, 1.570796, 1.696420],accel_mss,speed_ms,0,blend_radius_m)
    movel([0.124058, -1.393978, -2.547233, -0.771178, 1.570796, 1.694855],accel_mss,speed_ms,0,blend_radius_m)
    movel([0.122489, -1.393339, -2.547698, -0.771351, 1.570796, 1.693286],accel_mss,speed_ms,0,blend_radius_m)
    movel([0.120917, -1.392704, -2.548161, -0.771524, 1.570796, 1.691713],accel_mss,speed_ms,0,blend_radius_m)
    movel([0.119341, -1.392071, -2.548621, -0.771697, 1.570796, 1.690137],accel_mss,speed_ms,0,blend_radius_m)
    movel([0.117762, -1.391441, -2.549078, -0.771869, 1.570796, 1.688558],accel_mss,speed_ms,0,blend_radius_m)
    movel([0.116179, -1.390814, -2.549533, -0.772042, 1.570796, 1.686975],accel_mss,speed_ms,0,blend_radius_m)
    movel([0.114593, -1.390189, -2.549986, -0.772214, 1.570796, 1.685389],accel_mss,speed_ms,0,blend_radius_m)
    movel([0.113003, -1.389568, -2.550436, -0.772386, 1.570796, 1.683799],accel_mss,speed_ms,0,blend_radius_m)
    movel([0.111410, -1.388949, -2.550883, -0.772557, 1.570796, 1.682206],accel_mss,speed_ms,0,blend_radius_m)
    movel([0.109813, -1.388333, -2.551327, -0.772729, 1.570796, 1.680610],accel_mss,speed_ms,0,blend_radius_m)
    speed_ms = 0.005
    # Splitting Linear movement in 4 (instruction 233: MoveL 207)
    movel([0.109813, -1.390437, -2.552318, -0.769633, 1.570796, 1.680610],accel_mss,speed_ms,0,blend_radius_m)
    movel([0.109813, -1.392551, -2.553305, -0.766532, 1.570796, 1.680610],accel_mss,speed_ms,0,blend_radius_m)
    movel([0.109813, -1.394675, -2.554289, -0.763425, 1.570796, 1.680610],accel_mss,speed_ms,0,blend_radius_m)
    movel([0.109813, -1.396808, -2.555268, -0.760313, 1.570796, 1.680610],accel_mss,speed_ms,0,blend_radius_m)
    speed_ms = 0.035
    movel([0.111645, -1.397022, -2.555112, -0.760255, 1.570796, 1.682442],accel_mss,speed_ms,0,blend_radius_m)
    movel([0.112194, -1.397183, -2.554994, -0.760212, 1.570796, 1.682991],accel_mss,speed_ms,0,blend_radius_m)
    movel([0.112546, -1.397429, -2.554814, -0.760146, 1.570796, 1.683343],accel_mss,speed_ms,0,blend_radius_m)
    movel([0.112731, -1.397800, -2.554543, -0.760046, 1.570796, 1.683527],accel_mss,speed_ms,0,blend_radius_m)
    movel([0.112779, -1.398333, -2.554152, -0.759904, 1.570796, 1.683575],accel_mss,speed_ms,0,blend_radius_m)
    movel([0.112607, -1.400027, -2.552909, -0.759453, 1.570796, 1.683404],accel_mss,speed_ms,0,blend_radius_m)
    # Splitting Linear movement in 18 (instruction 241: MoveL 214)
    movel([0.112349, -1.402025, -2.551436, -0.758927, 1.570796, 1.683145],accel_mss,speed_ms,0,blend_radius_m)
    movel([0.112092, -1.404017, -2.549963, -0.758409, 1.570796, 1.682888],accel_mss,speed_ms,0,blend_radius_m)
    movel([0.111836, -1.406004, -2.548487, -0.757898, 1.570796, 1.682632],accel_mss,speed_ms,0,blend_radius_m)
    movel([0.111581, -1.407984, -2.547011, -0.757394, 1.570796, 1.682377],accel_mss,speed_ms,0,blend_radius_m)
    movel([0.111328, -1.409959, -2.545533, -0.756897, 1.570796, 1.682124],accel_mss,speed_ms,0,blend_radius_m)
    movel([0.111075, -1.411929, -2.544053, -0.756407, 1.570796, 1.681871],accel_mss,speed_ms,0,blend_radius_m)
    movel([0.110824, -1.413892, -2.542572, -0.755925, 1.570796, 1.681620],accel_mss,speed_ms,0,blend_radius_m)
    movel([0.110574, -1.415850, -2.541089, -0.755450, 1.570796, 1.681370],accel_mss,speed_ms,0,blend_radius_m)
    movel([0.110325, -1.417802, -2.539605, -0.754981, 1.570796, 1.681121],accel_mss,speed_ms,0,blend_radius_m)
    movel([0.110077, -1.419749, -2.538120, -0.754520, 1.570796, 1.680873],accel_mss,speed_ms,0,blend_radius_m)
    movel([0.109831, -1.421691, -2.536633, -0.754065, 1.570796, 1.680627],accel_mss,speed_ms,0,blend_radius_m)
    movel([0.109585, -1.423627, -2.535145, -0.753618, 1.570796, 1.680381],accel_mss,speed_ms,0,blend_radius_m)
    movel([0.109341, -1.425557, -2.533655, -0.753177, 1.570796, 1.680137],accel_mss,speed_ms,0,blend_radius_m)
    movel([0.109097, -1.427482, -2.532164, -0.752743, 1.570796, 1.679894],accel_mss,speed_ms,0,blend_radius_m)
    movel([0.108855, -1.429402, -2.530671, -0.752316, 1.570796, 1.679652],accel_mss,speed_ms,0,blend_radius_m)
    movel([0.108614, -1.431317, -2.529177, -0.751895, 1.570796, 1.679411],accel_mss,speed_ms,0,blend_radius_m)
    movel([0.108374, -1.433226, -2.527682, -0.751481, 1.570796, 1.679171],accel_mss,speed_ms,0,blend_radius_m)
    movel([0.108135, -1.435130, -2.526185, -0.751074, 1.570796, 1.678932],accel_mss,speed_ms,0,blend_radius_m)
    movel([0.107909, -1.436065, -2.525449, -0.750876, 1.570796, 1.678706],accel_mss,speed_ms,0,blend_radius_m)
    movel([0.107474, -1.436747, -2.524910, -0.750732, 1.570796, 1.678271],accel_mss,speed_ms,0,blend_radius_m)
    movel([0.107164, -1.436994, -2.524715, -0.750680, 1.570796, 1.677960],accel_mss,speed_ms,0,blend_radius_m)
    movel([0.106790, -1.437178, -2.524570, -0.750642, 1.570796, 1.677586],accel_mss,speed_ms,0,blend_radius_m)
    movel([0.105823, -1.437349, -2.524434, -0.750606, 1.570796, 1.676619],accel_mss,speed_ms,0,blend_radius_m)
    movel([0.105416, -1.437283, -2.524486, -0.750620, 1.570796, 1.676213],accel_mss,speed_ms,0,blend_radius_m)
    movel([0.105033, -1.437088, -2.524640, -0.750660, 1.570796, 1.675829],accel_mss,speed_ms,0,blend_radius_m)
    movel([0.104755, -1.436815, -2.524857, -0.750718, 1.570796, 1.675551],accel_mss,speed_ms,0,blend_radius_m)
    movel([0.104666, -1.436511, -2.525096, -0.750782, 1.570796, 1.675462],accel_mss,speed_ms,0,blend_radius_m)
    # Splitting Linear movement in 20 (instruction 251: MoveL 224)
    movel([0.104899, -1.434603, -2.526600, -0.751186, 1.570796, 1.675695],accel_mss,speed_ms,0,blend_radius_m)
    movel([0.105133, -1.432689, -2.528103, -0.751597, 1.570796, 1.675929],accel_mss,speed_ms,0,blend_radius_m)
    movel([0.105367, -1.430769, -2.529605, -0.752015, 1.570796, 1.676164],accel_mss,speed_ms,0,blend_radius_m)
    movel([0.105603, -1.428845, -2.531105, -0.752439, 1.570796, 1.676400],accel_mss,speed_ms,0,blend_radius_m)
    movel([0.105840, -1.426915, -2.532604, -0.752870, 1.570796, 1.676637],accel_mss,speed_ms,0,blend_radius_m)
    movel([0.106079, -1.424980, -2.534101, -0.753308, 1.570796, 1.676875],accel_mss,speed_ms,0,blend_radius_m)
    movel([0.106318, -1.423039, -2.535597, -0.753753, 1.570796, 1.677114],accel_mss,speed_ms,0,blend_radius_m)
    movel([0.106558, -1.421093, -2.537091, -0.754205, 1.570796, 1.677355],accel_mss,speed_ms,0,blend_radius_m)
    movel([0.106800, -1.419141, -2.538584, -0.754663, 1.570796, 1.677596],accel_mss,speed_ms,0,blend_radius_m)
    movel([0.107042, -1.417184, -2.540076, -0.755129, 1.570796, 1.677839],accel_mss,speed_ms,0,blend_radius_m)
    movel([0.107286, -1.415221, -2.541566, -0.755602, 1.570796, 1.678082],accel_mss,speed_ms,0,blend_radius_m)
    movel([0.107531, -1.413253, -2.543054, -0.756081, 1.570796, 1.678327],accel_mss,speed_ms,0,blend_radius_m)
    movel([0.107777, -1.411279, -2.544542, -0.756568, 1.570796, 1.678573],accel_mss,speed_ms,0,blend_radius_m)
    movel([0.108024, -1.409299, -2.546027, -0.757062, 1.570796, 1.678820],accel_mss,speed_ms,0,blend_radius_m)
    movel([0.108272, -1.407314, -2.547511, -0.757564, 1.570796, 1.679069],accel_mss,speed_ms,0,blend_radius_m)
    movel([0.108522, -1.405323, -2.548994, -0.758072, 1.570796, 1.679318],accel_mss,speed_ms,0,blend_radius_m)
    movel([0.108773, -1.403326, -2.550475, -0.758588, 1.570796, 1.679569],accel_mss,speed_ms,0,blend_radius_m)
    movel([0.109024, -1.401323, -2.551955, -0.759112, 1.570796, 1.679821],accel_mss,speed_ms,0,blend_radius_m)
    movel([0.109278, -1.399314, -2.553433, -0.759642, 1.570796, 1.680074],accel_mss,speed_ms,0,blend_radius_m)
    movel([0.109532, -1.397299, -2.554909, -0.760181, 1.570796, 1.680328],accel_mss,speed_ms,0,blend_radius_m)
    movel([0.109813, -1.396808, -2.555268, -0.760313, 1.570796, 1.680610],accel_mss,speed_ms,0,blend_radius_m)
    movel([0.111645, -1.397022, -2.555112, -0.760255, 1.570796, 1.682442],accel_mss,speed_ms,0,blend_radius_m)
    movel([0.111918, -1.397102, -2.555053, -0.760234, 1.570796, 1.682714],accel_mss,speed_ms,0,blend_radius_m)
    speed_ms = 0.005
    # Splitting Linear movement in 6 (instruction 256: MoveL 228)
    movel([0.111918, -1.395679, -2.554401, -0.762309, 1.570796, 1.682714],accel_mss,speed_ms,0,blend_radius_m)
    movel([0.111918, -1.394261, -2.553747, -0.764381, 1.570796, 1.682714],accel_mss,speed_ms,0,blend_radius_m)
    movel([0.111918, -1.392846, -2.553091, -0.766452, 1.570796, 1.682714],accel_mss,speed_ms,0,blend_radius_m)
    movel([0.111918, -1.391436, -2.552434, -0.768519, 1.570796, 1.682714],accel_mss,speed_ms,0,blend_radius_m)
    movel([0.111918, -1.390030, -2.551775, -0.770584, 1.570796, 1.682714],accel_mss,speed_ms,0,blend_radius_m)
    movel([0.111918, -1.388629, -2.551114, -0.772646, 1.570796, 1.682714],accel_mss,speed_ms,0,blend_radius_m)
    speed_ms = 0.040
    # Splitting Linear movement in 8 (instruction 258: MoveL 229)
    movel([0.112997, -1.386726, -2.552485, -0.773179, 1.570796, 1.683793],accel_mss,speed_ms,0,blend_radius_m)
    movel([0.114080, -1.384817, -2.553854, -0.773717, 1.570796, 1.684876],accel_mss,speed_ms,0,blend_radius_m)
    movel([0.115168, -1.382903, -2.555222, -0.774263, 1.570796, 1.685964],accel_mss,speed_ms,0,blend_radius_m)
    movel([0.116260, -1.380984, -2.556590, -0.774816, 1.570796, 1.687057],accel_mss,speed_ms,0,blend_radius_m)
    movel([0.117357, -1.379059, -2.557955, -0.775375, 1.570796, 1.688154],accel_mss,speed_ms,0,blend_radius_m)
    movel([0.118459, -1.377128, -2.559320, -0.775941, 1.570796, 1.689255],accel_mss,speed_ms,0,blend_radius_m)
    movel([0.119565, -1.375191, -2.560684, -0.776515, 1.570796, 1.690361],accel_mss,speed_ms,0,blend_radius_m)
    movel([0.120675, -1.373248, -2.562046, -0.777095, 1.570796, 1.691472],accel_mss,speed_ms,0,blend_radius_m)
    speed_ms = 0.005
    # Splitting Linear movement in 4 (instruction 260: MoveL 230)
    movel([0.120675, -1.375378, -2.563053, -0.773958, 1.570796, 1.691472],accel_mss,speed_ms,0,blend_radius_m)
    movel([0.120675, -1.377518, -2.564056, -0.770815, 1.570796, 1.691472],accel_mss,speed_ms,0,blend_radius_m)
    movel([0.120675, -1.379668, -2.565056, -0.767666, 1.570796, 1.691472],accel_mss,speed_ms,0,blend_radius_m)
    movel([0.120675, -1.381827, -2.566051, -0.764510, 1.570796, 1.691472],accel_mss,speed_ms,0,blend_radius_m)
    speed_ms = 0.035
    # Splitting Linear movement in 22 (instruction 262: MoveL 231)
    movel([0.122721, -1.382259, -2.565745, -0.764385, 1.570796, 1.693518],accel_mss,speed_ms,0,blend_radius_m)
    movel([0.124763, -1.382695, -2.565436, -0.764258, 1.570796, 1.695560],accel_mss,speed_ms,0,blend_radius_m)
    movel([0.126802, -1.383136, -2.565122, -0.764131, 1.570796, 1.697598],accel_mss,speed_ms,0,blend_radius_m)
    movel([0.128836, -1.383581, -2.564806, -0.764002, 1.570796, 1.699632],accel_mss,speed_ms,0,blend_radius_m)
    movel([0.130866, -1.384031, -2.564485, -0.763872, 1.570796, 1.701662],accel_mss,speed_ms,0,blend_radius_m)
    movel([0.132892, -1.384486, -2.564161, -0.763742, 1.570796, 1.703688],accel_mss,speed_ms,0,blend_radius_m)
    movel([0.134914, -1.384945, -2.563834, -0.763610, 1.570796, 1.705710],accel_mss,speed_ms,0,blend_radius_m)
    movel([0.136932, -1.385409, -2.563503, -0.763477, 1.570796, 1.707728],accel_mss,speed_ms,0,blend_radius_m)
    movel([0.138946, -1.385877, -2.563169, -0.763344, 1.570796, 1.709742],accel_mss,speed_ms,0,blend_radius_m)
    movel([0.140956, -1.386350, -2.562830, -0.763209, 1.570796, 1.711753],accel_mss,speed_ms,0,blend_radius_m)
    movel([0.142962, -1.386827, -2.562489, -0.763073, 1.570796, 1.713759],accel_mss,speed_ms,0,blend_radius_m)
    movel([0.144964, -1.387308, -2.562144, -0.762937, 1.570796, 1.715760],accel_mss,speed_ms,0,blend_radius_m)
    movel([0.146962, -1.387794, -2.561795, -0.762799, 1.570796, 1.717758],accel_mss,speed_ms,0,blend_radius_m)
    movel([0.148956, -1.388285, -2.561443, -0.762661, 1.570796, 1.719752],accel_mss,speed_ms,0,blend_radius_m)
    movel([0.150946, -1.388780, -2.561087, -0.762522, 1.570796, 1.721742],accel_mss,speed_ms,0,blend_radius_m)
    movel([0.152931, -1.389279, -2.560728, -0.762382, 1.570796, 1.723728],accel_mss,speed_ms,0,blend_radius_m)
    movel([0.154913, -1.389783, -2.560365, -0.762241, 1.570796, 1.725709],accel_mss,speed_ms,0,blend_radius_m)
    movel([0.156890, -1.390291, -2.559999, -0.762099, 1.570796, 1.727687],accel_mss,speed_ms,0,blend_radius_m)
    movel([0.158864, -1.390803, -2.559629, -0.761956, 1.570796, 1.729660],accel_mss,speed_ms,0,blend_radius_m)
    movel([0.160833, -1.391320, -2.559256, -0.761813, 1.570796, 1.731629],accel_mss,speed_ms,0,blend_radius_m)
    movel([0.162798, -1.391841, -2.558879, -0.761668, 1.570796, 1.733594],accel_mss,speed_ms,0,blend_radius_m)
    movel([0.164759, -1.392366, -2.558499, -0.761523, 1.570796, 1.735555],accel_mss,speed_ms,0,blend_radius_m)
    movel([0.166439, -1.392909, -2.558106, -0.761374, 1.570796, 1.737236],accel_mss,speed_ms,0,blend_radius_m)
    movel([0.167973, -1.393608, -2.557599, -0.761182, 1.570796, 1.738769],accel_mss,speed_ms,0,blend_radius_m)
    movel([0.169359, -1.394451, -2.556986, -0.760951, 1.570796, 1.740155],accel_mss,speed_ms,0,blend_radius_m)
    movel([0.170595, -1.395432, -2.556273, -0.760685, 1.570796, 1.741391],accel_mss,speed_ms,0,blend_radius_m)
    movel([0.171678, -1.396537, -2.555466, -0.760386, 1.570796, 1.742474],accel_mss,speed_ms,0,blend_radius_m)
    movel([0.172602, -1.397763, -2.554570, -0.760056, 1.570796, 1.743398],accel_mss,speed_ms,0,blend_radius_m)
    movel([0.173367, -1.399096, -2.553593, -0.759700, 1.570796, 1.744164],accel_mss,speed_ms,0,blend_radius_m)
    movel([0.173972, -1.400527, -2.552541, -0.759321, 1.570796, 1.744768],accel_mss,speed_ms,0,blend_radius_m)
    movel([0.174412, -1.402047, -2.551421, -0.758922, 1.570796, 1.745208],accel_mss,speed_ms,0,blend_radius_m)
    movel([0.174688, -1.403648, -2.550236, -0.758505, 1.570796, 1.745484],accel_mss,speed_ms,0,blend_radius_m)
    movel([0.174793, -1.405318, -2.548997, -0.758073, 1.570796, 1.745589],accel_mss,speed_ms,0,blend_radius_m)
    movel([0.174728, -1.407052, -2.547707, -0.757630, 1.570796, 1.745525],accel_mss,speed_ms,0,blend_radius_m)
    movel([0.174493, -1.408838, -2.546373, -0.757178, 1.570796, 1.745289],accel_mss,speed_ms,0,blend_radius_m)
    movel([0.174082, -1.410667, -2.545002, -0.756720, 1.570796, 1.744878],accel_mss,speed_ms,0,blend_radius_m)
    movel([0.173496, -1.412533, -2.543598, -0.756258, 1.570796, 1.744293],accel_mss,speed_ms,0,blend_radius_m)
    movel([0.172732, -1.414423, -2.542170, -0.755795, 1.570796, 1.743529],accel_mss,speed_ms,0,blend_radius_m)
    movel([0.171793, -1.416339, -2.540718, -0.755332, 1.570796, 1.742589],accel_mss,speed_ms,0,blend_radius_m)
    movel([0.170715, -1.418203, -2.539300, -0.754886, 1.570796, 1.741512],accel_mss,speed_ms,0,blend_radius_m)
    movel([0.169511, -1.420012, -2.537919, -0.754458, 1.570796, 1.740307],accel_mss,speed_ms,0,blend_radius_m)
    movel([0.168190, -1.421758, -2.536582, -0.754050, 1.570796, 1.738986],accel_mss,speed_ms,0,blend_radius_m)
    movel([0.166762, -1.423434, -2.535293, -0.753662, 1.570796, 1.737559],accel_mss,speed_ms,0,blend_radius_m)
    movel([0.165234, -1.425034, -2.534059, -0.753296, 1.570796, 1.736030],accel_mss,speed_ms,0,blend_radius_m)
    movel([0.163615, -1.426554, -2.532883, -0.752951, 1.570796, 1.734411],accel_mss,speed_ms,0,blend_radius_m)
    movel([0.161913, -1.427987, -2.531772, -0.752630, 1.570796, 1.732709],accel_mss,speed_ms,0,blend_radius_m)
    movel([0.160137, -1.429325, -2.530731, -0.752333, 1.570796, 1.730933],accel_mss,speed_ms,0,blend_radius_m)
    movel([0.158298, -1.430562, -2.529767, -0.752060, 1.570796, 1.729094],accel_mss,speed_ms,0,blend_radius_m)
    movel([0.156399, -1.431696, -2.528881, -0.751812, 1.570796, 1.727195],accel_mss,speed_ms,0,blend_radius_m)
    movel([0.154454, -1.432719, -2.528080, -0.751590, 1.570796, 1.725250],accel_mss,speed_ms,0,blend_radius_m)
    movel([0.152467, -1.433622, -2.527371, -0.751396, 1.570796, 1.723263],accel_mss,speed_ms,0,blend_radius_m)
    movel([0.150445, -1.434402, -2.526758, -0.751229, 1.570796, 1.721242],accel_mss,speed_ms,0,blend_radius_m)
    movel([0.148397, -1.435054, -2.526245, -0.751090, 1.570796, 1.719194],accel_mss,speed_ms,0,blend_radius_m)
    movel([0.146334, -1.435567, -2.525841, -0.750981, 1.570796, 1.717131],accel_mss,speed_ms,0,blend_radius_m)
    # Splitting Linear movement in 28 (instruction 295: MoveL 264)
    movel([0.144149, -1.436037, -2.525470, -0.750882, 1.570796, 1.714945],accel_mss,speed_ms,0,blend_radius_m)
    movel([0.141963, -1.436511, -2.525097, -0.750782, 1.570796, 1.712760],accel_mss,speed_ms,0,blend_radius_m)
    movel([0.139779, -1.436988, -2.524720, -0.750682, 1.570796, 1.710575],accel_mss,speed_ms,0,blend_radius_m)
    movel([0.137595, -1.437468, -2.524340, -0.750581, 1.570796, 1.708391],accel_mss,speed_ms,0,blend_radius_m)
    movel([0.135412, -1.437952, -2.523957, -0.750480, 1.570796, 1.706208],accel_mss,speed_ms,0,blend_radius_m)
    movel([0.133229, -1.438439, -2.523571, -0.750379, 1.570796, 1.704025],accel_mss,speed_ms,0,blend_radius_m)
    movel([0.131047, -1.438930, -2.523182, -0.750277, 1.570796, 1.701843],accel_mss,speed_ms,0,blend_radius_m)
    movel([0.128865, -1.439424, -2.522790, -0.750175, 1.570796, 1.699662],accel_mss,speed_ms,0,blend_radius_m)
    movel([0.126685, -1.439921, -2.522395, -0.750073, 1.570796, 1.697481],accel_mss,speed_ms,0,blend_radius_m)
    movel([0.124505, -1.440422, -2.521997, -0.749970, 1.570796, 1.695301],accel_mss,speed_ms,0,blend_radius_m)
    movel([0.122325, -1.440926, -2.521596, -0.749867, 1.570796, 1.693122],accel_mss,speed_ms,0,blend_radius_m)
    movel([0.120147, -1.441433, -2.521191, -0.749764, 1.570796, 1.690943],accel_mss,speed_ms,0,blend_radius_m)
    movel([0.117969, -1.441944, -2.520784, -0.749661, 1.570796, 1.688765],accel_mss,speed_ms,0,blend_radius_m)
    movel([0.115792, -1.442458, -2.520374, -0.749557, 1.570796, 1.686588],accel_mss,speed_ms,0,blend_radius_m)
    movel([0.113616, -1.442975, -2.519961, -0.749453, 1.570796, 1.684412],accel_mss,speed_ms,0,blend_radius_m)
    movel([0.111441, -1.443496, -2.519544, -0.749349, 1.570796, 1.682237],accel_mss,speed_ms,0,blend_radius_m)
    movel([0.109266, -1.444020, -2.519125, -0.749244, 1.570796, 1.680063],accel_mss,speed_ms,0,blend_radius_m)
    movel([0.107093, -1.444547, -2.518703, -0.749140, 1.570796, 1.677889],accel_mss,speed_ms,0,blend_radius_m)
    movel([0.104920, -1.445077, -2.518277, -0.749035, 1.570796, 1.675716],accel_mss,speed_ms,0,blend_radius_m)
    movel([0.102748, -1.445610, -2.517849, -0.748930, 1.570796, 1.673545],accel_mss,speed_ms,0,blend_radius_m)
    movel([0.100577, -1.446147, -2.517418, -0.748824, 1.570796, 1.671374],accel_mss,speed_ms,0,blend_radius_m)
    movel([0.098407, -1.446687, -2.516984, -0.748719, 1.570796, 1.669204],accel_mss,speed_ms,0,blend_radius_m)
    movel([0.096238, -1.447230, -2.516546, -0.748613, 1.570796, 1.667035],accel_mss,speed_ms,0,blend_radius_m)
    movel([0.094070, -1.447776, -2.516106, -0.748507, 1.570796, 1.664867],accel_mss,speed_ms,0,blend_radius_m)
    movel([0.091903, -1.448325, -2.515663, -0.748401, 1.570796, 1.662700],accel_mss,speed_ms,0,blend_radius_m)
    movel([0.089738, -1.448877, -2.515216, -0.748295, 1.570796, 1.660534],accel_mss,speed_ms,0,blend_radius_m)
    movel([0.087573, -1.449433, -2.514767, -0.748189, 1.570796, 1.658369],accel_mss,speed_ms,0,blend_radius_m)
    movel([0.085409, -1.449991, -2.514315, -0.748083, 1.570796, 1.656205],accel_mss,speed_ms,0,blend_radius_m)
    movel([0.083905, -1.450402, -2.513982, -0.748005, 1.570796, 1.654702],accel_mss,speed_ms,0,blend_radius_m)
    movel([0.083590, -1.450384, -2.513997, -0.748008, 1.570796, 1.654387],accel_mss,speed_ms,0,blend_radius_m)
    movel([0.083340, -1.450250, -2.514105, -0.748034, 1.570796, 1.654136],accel_mss,speed_ms,0,blend_radius_m)
    movel([0.083173, -1.449969, -2.514333, -0.748087, 1.570796, 1.653970],accel_mss,speed_ms,0,blend_radius_m)
    movel([0.083159, -1.448950, -2.515157, -0.748281, 1.570796, 1.653955],accel_mss,speed_ms,0,blend_radius_m)
    movel([0.083312, -1.448505, -2.515517, -0.748367, 1.570796, 1.654109],accel_mss,speed_ms,0,blend_radius_m)
    movel([0.083555, -1.448156, -2.515799, -0.748434, 1.570796, 1.654351],accel_mss,speed_ms,0,blend_radius_m)
    movel([0.083875, -1.447888, -2.516015, -0.748486, 1.570796, 1.654671],accel_mss,speed_ms,0,blend_radius_m)
    movel([0.084695, -1.447516, -2.516315, -0.748558, 1.570796, 1.655492],accel_mss,speed_ms,0,blend_radius_m)
    movel([0.085672, -1.447246, -2.516533, -0.748610, 1.570796, 1.656468],accel_mss,speed_ms,0,blend_radius_m)
    # Splitting Linear movement in 26 (instruction 306: MoveL 275)
    movel([0.087929, -1.446662, -2.517003, -0.748724, 1.570796, 1.658725],accel_mss,speed_ms,0,blend_radius_m)
    movel([0.090187, -1.446081, -2.517471, -0.748837, 1.570796, 1.660983],accel_mss,speed_ms,0,blend_radius_m)
    movel([0.092446, -1.445504, -2.517935, -0.748951, 1.570796, 1.663242],accel_mss,speed_ms,0,blend_radius_m)
    movel([0.094706, -1.444929, -2.518396, -0.749064, 1.570796, 1.665502],accel_mss,speed_ms,0,blend_radius_m)
    movel([0.096967, -1.444359, -2.518854, -0.749177, 1.570796, 1.667764],accel_mss,speed_ms,0,blend_radius_m)
    movel([0.099230, -1.443791, -2.519308, -0.749290, 1.570796, 1.670026],accel_mss,speed_ms,0,blend_radius_m)
    movel([0.101493, -1.443227, -2.519759, -0.749403, 1.570796, 1.672290],accel_mss,speed_ms,0,blend_radius_m)
    movel([0.103758, -1.442667, -2.520207, -0.749515, 1.570796, 1.674554],accel_mss,speed_ms,0,blend_radius_m)
    movel([0.106023, -1.442110, -2.520652, -0.749627, 1.570796, 1.676819],accel_mss,speed_ms,0,blend_radius_m)
    movel([0.108289, -1.441556, -2.521093, -0.749739, 1.570796, 1.679086],accel_mss,speed_ms,0,blend_radius_m)
    movel([0.110557, -1.441006, -2.521532, -0.749851, 1.570796, 1.681353],accel_mss,speed_ms,0,blend_radius_m)
    movel([0.112825, -1.440460, -2.521967, -0.749963, 1.570796, 1.683621],accel_mss,speed_ms,0,blend_radius_m)
    movel([0.115094, -1.439917, -2.522398, -0.750074, 1.570796, 1.685891],accel_mss,speed_ms,0,blend_radius_m)
    movel([0.117364, -1.439377, -2.522827, -0.750185, 1.570796, 1.688161],accel_mss,speed_ms,0,blend_radius_m)
    movel([0.119635, -1.438842, -2.523252, -0.750295, 1.570796, 1.690432],accel_mss,speed_ms,0,blend_radius_m)
    movel([0.121907, -1.438309, -2.523674, -0.750406, 1.570796, 1.692704],accel_mss,speed_ms,0,blend_radius_m)
    movel([0.124180, -1.437781, -2.524093, -0.750516, 1.570796, 1.694976],accel_mss,speed_ms,0,blend_radius_m)
    movel([0.126453, -1.437256, -2.524508, -0.750625, 1.570796, 1.697250],accel_mss,speed_ms,0,blend_radius_m)
    movel([0.128728, -1.436734, -2.524920, -0.750735, 1.570796, 1.699524],accel_mss,speed_ms,0,blend_radius_m)
    movel([0.131003, -1.436216, -2.525329, -0.750844, 1.570796, 1.701799],accel_mss,speed_ms,0,blend_radius_m)
    movel([0.133279, -1.435702, -2.525734, -0.750952, 1.570796, 1.704075],accel_mss,speed_ms,0,blend_radius_m)
    movel([0.135555, -1.435192, -2.526137, -0.751061, 1.570796, 1.706351],accel_mss,speed_ms,0,blend_radius_m)
    movel([0.137832, -1.434685, -2.526535, -0.751168, 1.570796, 1.708629],accel_mss,speed_ms,0,blend_radius_m)
    movel([0.140110, -1.434182, -2.526931, -0.751276, 1.570796, 1.710906],accel_mss,speed_ms,0,blend_radius_m)
    movel([0.142389, -1.433683, -2.527323, -0.751383, 1.570796, 1.713185],accel_mss,speed_ms,0,blend_radius_m)
    movel([0.144668, -1.433187, -2.527712, -0.751489, 1.570796, 1.715464],accel_mss,speed_ms,0,blend_radius_m)
    movel([0.146571, -1.432737, -2.528066, -0.751587, 1.570796, 1.717367],accel_mss,speed_ms,0,blend_radius_m)
    movel([0.148451, -1.432204, -2.528483, -0.751702, 1.570796, 1.719247],accel_mss,speed_ms,0,blend_radius_m)
    movel([0.150313, -1.431577, -2.528974, -0.751838, 1.570796, 1.721109],accel_mss,speed_ms,0,blend_radius_m)
    movel([0.152157, -1.430846, -2.529545, -0.751998, 1.570796, 1.722953],accel_mss,speed_ms,0,blend_radius_m)
    movel([0.153985, -1.429998, -2.530207, -0.752184, 1.570796, 1.724781],accel_mss,speed_ms,0,blend_radius_m)
    movel([0.155798, -1.429026, -2.530964, -0.752399, 1.570796, 1.726594],accel_mss,speed_ms,0,blend_radius_m)
    movel([0.157601, -1.427912, -2.531830, -0.752647, 1.570796, 1.728398],accel_mss,speed_ms,0,blend_radius_m)
    movel([0.159392, -1.426651, -2.532808, -0.752930, 1.570796, 1.730189],accel_mss,speed_ms,0,blend_radius_m)
    movel([0.161799, -1.424676, -2.534335, -0.753377, 1.570796, 1.732595],accel_mss,speed_ms,0,blend_radius_m)
    movel([0.163946, -1.422580, -2.535950, -0.753859, 1.570796, 1.734742],accel_mss,speed_ms,0,blend_radius_m)
    movel([0.165825, -1.420386, -2.537633, -0.754370, 1.570796, 1.736622],accel_mss,speed_ms,0,blend_radius_m)
    movel([0.167436, -1.418119, -2.539364, -0.754906, 1.570796, 1.738232],accel_mss,speed_ms,0,blend_radius_m)
    movel([0.168771, -1.415806, -2.541122, -0.755460, 1.570796, 1.739568],accel_mss,speed_ms,0,blend_radius_m)
    movel([0.169823, -1.413480, -2.542883, -0.756026, 1.570796, 1.740619],accel_mss,speed_ms,0,blend_radius_m)
    movel([0.170587, -1.411163, -2.544629, -0.756597, 1.570796, 1.741383],accel_mss,speed_ms,0,blend_radius_m)
    movel([0.171055, -1.408889, -2.546334, -0.757165, 1.570796, 1.741851],accel_mss,speed_ms,0,blend_radius_m)
    movel([0.171221, -1.406685, -2.547981, -0.757724, 1.570796, 1.742017],accel_mss,speed_ms,0,blend_radius_m)
    movel([0.171077, -1.404580, -2.549545, -0.758263, 1.570796, 1.741873],accel_mss,speed_ms,0,blend_radius_m)
    movel([0.170618, -1.402609, -2.551005, -0.758775, 1.570796, 1.741414],accel_mss,speed_ms,0,blend_radius_m)
    movel([0.169835, -1.400800, -2.552340, -0.759249, 1.570796, 1.740631],accel_mss,speed_ms,0,blend_radius_m)
    movel([0.168721, -1.399189, -2.553525, -0.759676, 1.570796, 1.739517],accel_mss,speed_ms,0,blend_radius_m)
    movel([0.167272, -1.397802, -2.554541, -0.760046, 1.570796, 1.738068],accel_mss,speed_ms,0,blend_radius_m)
    movel([0.165480, -1.396676, -2.555365, -0.760348, 1.570796, 1.736276],accel_mss,speed_ms,0,blend_radius_m)
    movel([0.163342, -1.395840, -2.555975, -0.760574, 1.570796, 1.734139],accel_mss,speed_ms,0,blend_radius_m)
    # Splitting Linear movement in 6 (instruction 331: MoveL 300)
    movel([0.161964, -1.395450, -2.556260, -0.760680, 1.570796, 1.732760],accel_mss,speed_ms,0,blend_radius_m)
    movel([0.160583, -1.395061, -2.556543, -0.760786, 1.570796, 1.731379],accel_mss,speed_ms,0,blend_radius_m)
    movel([0.159200, -1.394674, -2.556824, -0.760891, 1.570796, 1.729996],accel_mss,speed_ms,0,blend_radius_m)
    movel([0.157815, -1.394290, -2.557104, -0.760996, 1.570796, 1.728611],accel_mss,speed_ms,0,blend_radius_m)
    movel([0.156427, -1.393907, -2.557382, -0.761100, 1.570796, 1.727224],accel_mss,speed_ms,0,blend_radius_m)
    movel([0.155038, -1.393527, -2.557658, -0.761204, 1.570796, 1.725834],accel_mss,speed_ms,0,blend_radius_m)
    # Splitting Linear movement in 18 (instruction 332: MoveL 301)
    movel([0.153192, -1.393056, -2.557999, -0.761333, 1.570796, 1.723988],accel_mss,speed_ms,0,blend_radius_m)
    movel([0.151342, -1.392590, -2.558337, -0.761462, 1.570796, 1.722138],accel_mss,speed_ms,0,blend_radius_m)
    movel([0.149489, -1.392127, -2.558673, -0.761589, 1.570796, 1.720285],accel_mss,speed_ms,0,blend_radius_m)
    movel([0.147632, -1.391668, -2.559005, -0.761716, 1.570796, 1.718428],accel_mss,speed_ms,0,blend_radius_m)
    movel([0.145771, -1.391213, -2.559334, -0.761842, 1.570796, 1.716568],accel_mss,speed_ms,0,blend_radius_m)
    movel([0.143907, -1.390762, -2.559660, -0.761968, 1.570796, 1.714704],accel_mss,speed_ms,0,blend_radius_m)
    movel([0.142040, -1.390314, -2.559982, -0.762092, 1.570796, 1.712836],accel_mss,speed_ms,0,blend_radius_m)
    movel([0.140169, -1.389871, -2.560302, -0.762216, 1.570796, 1.710965],accel_mss,speed_ms,0,blend_radius_m)
    movel([0.138294, -1.389431, -2.560619, -0.762339, 1.570796, 1.709091],accel_mss,speed_ms,0,blend_radius_m)
    movel([0.136416, -1.388995, -2.560933, -0.762461, 1.570796, 1.707213],accel_mss,speed_ms,0,blend_radius_m)
    movel([0.134535, -1.388563, -2.561243, -0.762583, 1.570796, 1.705331],accel_mss,speed_ms,0,blend_radius_m)
    movel([0.132650, -1.388135, -2.561550, -0.762703, 1.570796, 1.703446],accel_mss,speed_ms,0,blend_radius_m)
    movel([0.130761, -1.387711, -2.561855, -0.762823, 1.570796, 1.701558],accel_mss,speed_ms,0,blend_radius_m)
